(* IEC 61131-3 sources: beebread/doc (part 2) *)

FUNCTION WORD_TO_RANGE : REAL
VAR_INPUT
	X : WORD;
	low : REAL;
	high : REAL;
END_VAR

WORD_TO_RANGE := (high - low) * WORD_TO_REAL(X) * 0.00001525902189669640 + low;
END_FUNCTION

// Commented out for beedance: it uses CHR_TO_STRING, which is commented out.
// FUNCTION LIST_ADD : BOOL
// VAR_INPUT
// 	SEP : BYTE;
// 	INS : STRING(LIST_LENGTH);
// END_VAR
// VAR_IN_OUT
// 	LIST : STRING(LIST_LENGTH);
// END_VAR
// VAR
// 	sx : STRING(1);
// END_VAR
// VAR
// 	INS_work : STRING;
// END_VAR
// (* IEC 61131-3 does not let a POU assign to its inputs, so the body works on copies. *)
// INS_work := INS;
//
// sx := CHR_TO_STRING(SEP);			(* convert separation character to string *)
// INS_work := CONCAT(sx, INS_work);					(* start element with separation character *)
//
// IF LEN(LIST) + LEN(INS_work) > LIST_LENGTH THEN
// 	LIST_ADD := FALSE;					(* return false if element does not fit *)
// ELSE
// 	LIST := CONCAT(LIST, INS_work);
// 	LIST_ADD := TRUE;
// END_IF;
// END_FUNCTION

// Commented out for beedance: it reads or writes the bytes of a STRING through a pointer; a beedance reference (REF_TO) refers to a whole variable of its type.
// FUNCTION LIST_CLEAN : BOOL
// VAR_INPUT
// 	SEP : BYTE;
// END_VAR
// VAR_IN_OUT
// 	LIST : STRING(LIST_LENGTH);
// END_VAR
// VAR
// 	pt : REF_TO ARRAY[1..LIST_LENGTH] OF BYTE;
// 	read : INT := 1;
// 	write : INT := 1;
// 	last: BYTE;
// 	c: BYTE;
// END_VAR
//
// pt := REF(LIST);
//
// FOR read := 1 TO LIST_LENGTH DO
// 	c := pt^[read];								(* read character from list *)
// 	IF c = 0 THEN EXIT;						(* exit the loop if character definbes end of string *)
// 	ELSIF c <> SEP OR sep <> last THEN	(* copy element from read to write position unless a double sep character is present *)
// 		pt^[write] := c;
// 		write := write + 1;
// 	END_IF;
// 	last := c;									(* remember last character *)
// END_FOR;
//
// IF last = SEP THEN write := write - 1; END_IF;		(* if last character is sep then delete empty element at end *)
// IF write <= STRING_LENGTH THEN pt^[write] := 0;	 END_IF;		(* terminate string with 0 *)
//
// LIST_CLEAN := TRUE;						(* retrun TRUE *)
// END_FUNCTION

// Commented out for beedance: it reads or writes the bytes of a STRING through a pointer; a beedance reference (REF_TO) refers to a whole variable of its type.
// FUNCTION LIST_GET : STRING(LIST_LENGTH)
// VAR_INPUT
// 	SEP : BYTE;
// 	POS : INT;
// END_VAR
// VAR_IN_OUT
// 	LIST : STRING(LIST_LENGTH);
// END_VAR
// VAR
// 	i : INT := 1;
// 	o : INT := 1;
// 	pt : REF_TO ARRAY[1..LIST_LENGTH] OF BYTE;
// 	po : REF_TO ARRAY[1..LIST_LENGTH] OF BYTE;
// 	cnt: INT := 0;
// 	c: BYTE;
// END_VAR
//
// pt := REF(LIST);							(* load pointers *)
// po := REF(LIST_GET);
//
// REPEAT
// 	c := pt^[i];
// 	IF cnt = pos THEN						(* copy element to output string *)
// 		IF c = SEP  THEN EXIT; END_IF;		(* next element stop copy and finish *)
// 		po^[o] := c;
// 		o := o + 1;
// 	ELSIF c = SEP THEN
// 		cnt := cnt + 1;
// 	END_IF;
// 	i := i + 1;
// UNTIL
// 	(i = LIST_LENGTH) OR (c = 0)
// END_REPEAT;
// po^[o] := 0;						(* close the output string *)
// END_FUNCTION

// Commented out for beedance: it reads or writes the bytes of a STRING through a pointer; a beedance reference (REF_TO) refers to a whole variable of its type.
// FUNCTION LIST_INSERT : BOOL
// VAR_INPUT
// 	SEP : BYTE;
// 	POS : INT;
// 	INS : STRING(LIST_LENGTH);
// END_VAR
// VAR_IN_OUT
// 	LIST : STRING(LIST_LENGTH);
// END_VAR
// VAR
// 	pt : REF_TO ARRAY[1..LIST_LENGTH] OF BYTE;
// 	read : INT := 1;
// 	cnt : INT := 1;
// 	sx : STRING(1);
// END_VAR
//
// (* load pointers *)
// pt := REF(LIST);
//
// IF LEN(ins) + 1 + LEN(LIST) > LIST_LENGTH THEN
// 	LIST_INSERT := FALSE;
// ELSE
// 	LIST_INSERT := TRUE;
// 	(* search for position *)
// 	WHILE read < LIST_LENGTH DO
// 		IF cnt >= POS THEN
// 			sx := CHR_TO_STRING(SEP);
// 			INS := CONCAT(sx, INS);
// 			LIST := INSERT(LIST, INS, read - 1);
// 			LIST_INSERT := TRUE;
// 			RETURN;
// 		END_IF;
// 		IF pt^[read]  = 0 THEN				(* list is too short add empty element *)
// 			pt^[read] := SEP;
// 			pt^[read + 1] := 0;
// 		END_IF;
// 		read := read + 1;
// 		IF pt^[read] = SEP OR pt^[read] = 0 THEN cnt := cnt + 1; END_IF;
// 	END_WHILE;
// END_IF;
// END_FUNCTION

// Commented out for beedance: it reads or writes the bytes of a STRING through a pointer; a beedance reference (REF_TO) refers to a whole variable of its type.
// FUNCTION LIST_LEN : INT
// VAR_INPUT
// 	SEP : BYTE;
// END_VAR
// VAR_IN_OUT
// 	LIST : STRING(LIST_LENGTH);
// END_VAR
// VAR
// 	pt : REF_TO ARRAY[1..LIST_LENGTH] OF BYTE;
// 	pos: INT := 1;
// 	c: BYTE;
// END_VAR
//
// pt := REF(LIST);
// LIST_LEN := 0;
// REPEAT
// 	c := pt^[pos];
// 	IF c = SEP THEN LIST_LEN := LIST_LEN + 1; END_IF;
// 	pos := pos + 1;
// UNTIL
// 	c = 0 OR pos > LIST_LENGTH
// END_REPEAT;
// END_FUNCTION

// Commented out for beedance: it reads or writes the bytes of a STRING through a pointer; a beedance reference (REF_TO) refers to a whole variable of its type.
// FUNCTION_BLOCK LIST_NEXT
// VAR_INPUT
// 	SEP : BYTE;
// 	RST : BOOL;
// END_VAR
// VAR_IN_OUT
// 	LIST : STRING(LIST_LENGTH);
// END_VAR
// VAR_OUTPUT
// 	LEL : STRING(LIST_LENGTH);
// 	NUL : BOOL;
// END_VAR
// VAR
// 	pos : INT := 1;
// 	pt : REF_TO ARRAY[1..LIST_LENGTH] OF BYTE;
// 	po : REF_TO ARRAY[1..LIST_LENGTH] OF BYTE;
// 	c: BYTE;
// 	write: INT;
// END_VAR
//
// pt := REF(LIST);
// po := REF(LEL);
//
// IF rst THEN
// 	pos := 1;
// END_IF;
//
// IF pt^[pos] = 0 OR pos = LIST_LENGTH THEN
// 	LEL := '';
// 	NUL := TRUE;
// ELSE
// 	NUL := FALSE;
// 	write := 1;
// 	FOR pos := pos + 1 TO LIST_LENGTH DO
// 		c := pt^[pos];
// 		IF c = 0 OR c = SEP THEN
// 			po^[write] := 0;
// 			RETURN;
// 		ELSE
// 			po^[write] := pt^[pos];
// 			write := write + 1;
// 		END_IF;
// 	END_FOR;
// END_IF;
// END_FUNCTION_BLOCK

// Commented out for beedance: it reads or writes the bytes of a STRING through a pointer; a beedance reference (REF_TO) refers to a whole variable of its type.
// FUNCTION LIST_RETRIEVE : STRING(LIST_LENGTH)
// VAR_INPUT
// 	SEP : BYTE;
// 	POS : INT;
// END_VAR
// VAR_IN_OUT
// 	LIST : STRING(LIST_LENGTH);
// END_VAR
// VAR
// 	i :	INT;
// 	o : INT := 1;
// 	w : INT := 1;
// 	pt : REF_TO ARRAY[1..LIST_LENGTH] OF BYTE;
// 	po : REF_TO ARRAY[1..LIST_LENGTH] OF BYTE;
// 	cnt: INT := 0;
// 	c: BYTE;
// END_VAR
//
// (* load pointers *)
// pt := REF(LIST);
// po := REF(LIST_RETRIEVE);
//
// IF pos > 0 THEN
// 	FOR i := 1 TO LIST_LENGTH DO
// 		c := pt^[i];
// 		IF c = 0 THEN
// 			po^[o] := 0;
// 			IF cnt < pos THEN pt^[w + 1] := 0; ELSE pt^[w] := 0; END_IF;
// 			RETURN;
// 		ELSIF cnt = pos AND c <> SEP THEN				(* we have found the element *)
// 			po^[o] := pt^[i];
// 			o := o + 1;
// 		ELSIF cnt >= pos THEN
// 			pt^[w] := c;
// 			w := w + 1;
// 		ELSE
// 			w := i;
// 		END_IF;
// 		IF c = sep THEN cnt := cnt + 1; END_IF;
// 	END_FOR;
// ELSE
// 	LIST_RETRIEVE := '';
// END_IF;
// END_FUNCTION

// Commented out for beedance: it reads or writes the bytes of a STRING through a pointer; a beedance reference (REF_TO) refers to a whole variable of its type.
// FUNCTION LIST_RETRIEVE_LAST : STRING(LIST_LENGTH)
// VAR_INPUT
// 	SEP : BYTE;
// END_VAR
// VAR_IN_OUT
// 	LIST : STRING(LIST_LENGTH);
// END_VAR
// VAR
// 	i :	INT;
// 	last : INT := 1;
// 	pt : REF_TO ARRAY[1..LIST_LENGTH] OF BYTE;
// 	c: BYTE;
// END_VAR
//
// (* load pointers *)
// pt := REF(LIST);
//
// (* search position of last element *)
// FOR i := 1 TO LIST_LENGTH DO
// 	c := pt^[i];
// 	IF c = 0 THEN
// 		EXIT;
// 	ELSIF C = SEP THEN
// 		last := i;
// 	END_IF;
// END_FOR;
// (* return last element of list *)
// LIST_RETRIEVE_LAST := MID(LIST, LIST_LENGTH, last + 1);
// (* terminate list at i *)
// pt^[last] := 0;
// END_FUNCTION

FUNCTION_BLOCK COUNT_BR
VAR_INPUT
	SET : BOOL;
	IN : BYTE;
	UP : BOOL;
	DN : BOOL;
	STEP : BYTE := 1;
	MX : BYTE := 255;
	RST : BOOL;
END_VAR
VAR_OUTPUT
	CNT : BYTE;
END_VAR
VAR
	last_up: BOOL;
	last_dn: BOOL;
END_VAR

IF rst THEN
	cnt := 0;
ELSIF set THEN
	cnt := LIMIT(0,in,mx);
ELSIF up AND NOT last_up THEN
	cnt := INT_TO_BYTE(INC(cnt,step,mx));
ELSIF dn AND NOT last_dn THEN
	cnt := INT_TO_BYTE(inc(cnt,-step,mx));
END_IF;
last_up := up;
last_dn := dn;
END_FUNCTION_BLOCK

FUNCTION_BLOCK COUNT_DR
VAR_INPUT
	SET : BOOL;
	IN : DWORD;
	UP : BOOL;
	DN : BOOL;
	STEP : DWORD := 1;
	MX : DWORD := 16#FFFFFFFF;
	RST : BOOL;
END_VAR
VAR_OUTPUT
	CNT : DWORD;
END_VAR
VAR
	last_up: BOOL;
	last_dn: BOOL;
END_VAR

IF rst THEN
	cnt := 0;
ELSIF set THEN
	cnt := LIMIT(DWORD#0,in,mx);
ELSIF up AND NOT last_up THEN
	IF STEP > ULINT_TO_DWORD((DWORD_TO_ULINT(MX) + 4294967296 - DWORD_TO_ULINT(CNT)) MOD 4294967296) THEN
		CNT := ULINT_TO_DWORD((DWORD_TO_ULINT(CNT) + 4294967296 - DWORD_TO_ULINT(MX) + DWORD_TO_ULINT(STEP) - 1) MOD 4294967296);
	ELSE
		CNT := ULINT_TO_DWORD((DWORD_TO_ULINT(CNT) + DWORD_TO_ULINT(STEP)) MOD 4294967296);
	END_IF;
ELSIF dn AND NOT last_dn THEN
	IF STEP > CNT THEN
		CNT := ULINT_TO_DWORD((DWORD_TO_ULINT(CNT) + 4294967296 - DWORD_TO_ULINT(STEP) + DWORD_TO_ULINT(MX) + 1) MOD 4294967296);
	ELSE
		CNT := ULINT_TO_DWORD((DWORD_TO_ULINT(CNT) + 4294967296 - DWORD_TO_ULINT(STEP)) MOD 4294967296);
	END_IF;
END_IF;
last_up := up;
last_dn := dn;
END_FUNCTION_BLOCK

FUNCTION_BLOCK FF_D2E
VAR_INPUT
	D0 : BOOL;
	D1 : BOOL;
	CLK : BOOL;
	RST : BOOL;
END_VAR
VAR_OUTPUT
	Q0 : BOOL;
	Q1 : BOOL;
END_VAR
VAR
	edge : BOOL;
END_VAR

IF rst THEN
	Q0 := FALSE;
	Q1 := FALSE;
ELSIF clk AND NOT edge THEN
	Q0 := D0;
	Q1 := D1;
END_IF;
edge := CLK;
END_FUNCTION_BLOCK

FUNCTION_BLOCK FF_D4E
VAR_INPUT
	D0 : BOOL;
	D1 : BOOL;
	D2 : BOOL;
	D3 : BOOL;
	CLK : BOOL;
	RST : BOOL;
END_VAR
VAR_OUTPUT
	Q0 : BOOL;
	Q1 : BOOL;
	Q2 : BOOL;
	Q3 : BOOL;
END_VAR
VAR
	edge : BOOL;
END_VAR

IF rst THEN
	Q0 := FALSE;
	Q1 := FALSE;
	Q2 := FALSE;
	Q3 := FALSE;
ELSIF clk AND NOT edge THEN
	Q0 := D0;
	Q1 := D1;
	Q2 := D2;
	Q3 := D3;
END_IF;
edge := CLK;
END_FUNCTION_BLOCK

FUNCTION_BLOCK FF_DRE
VAR_INPUT
	SET : BOOL;
	D : BOOL;
	CLK : BOOL;
	RST : BOOL;
END_VAR
VAR_OUTPUT
	Q : BOOL;
END_VAR
VAR
	edge : BOOL;
END_VAR

IF rst OR set THEN
	Q := NOT rst;
ELSIF clk AND NOT edge THEN
	Q := D;
END_IF;
edge := CLK;
END_FUNCTION_BLOCK

FUNCTION_BLOCK FF_JKE
VAR_INPUT
	SET : BOOL;
	J : BOOL;
	CLK : BOOL;
	K : BOOL;
	RST : BOOL;
END_VAR
VAR_OUTPUT
	Q : BOOL;
END_VAR
VAR
	edge : BOOL;
END_VAR

IF rst OR set THEN
	Q := NOT rst;
ELSIF clk AND NOT edge THEN
	IF J XOR K THEN Q := J;
	ELSE Q := K XOR Q;
	END_IF;
END_IF;
edge := CLK;
END_FUNCTION_BLOCK

FUNCTION_BLOCK FF_RSE
VAR_INPUT
	CS : BOOL;
	CR : BOOL;
	RST : BOOL;
END_VAR
VAR_OUTPUT
	Q : BOOL;
END_VAR
VAR
	es, er : BOOL;
END_VAR

IF rst THEN
	(* asynchronous reset *)
	Q := FALSE;
ELSIF CR AND NOT er THEN
	(* rising edge on CR *)
	Q := FALSE;
ELSIF CS AND NOT es THEN
	(* rising edge on CS *)
	Q := TRUE;
END_IF;

es := CS;
er := CR;
END_FUNCTION_BLOCK

FUNCTION_BLOCK SELECT_8
VAR_INPUT
	E : BOOL;
	SET : BOOL;
	IN : BYTE;
	UP : BOOL;
	DN : BOOL;
	RST : BOOL;
END_VAR
VAR_OUTPUT
	Q0, Q1, Q2, Q3, Q4, Q5, Q6, Q7 : BOOL;
	STATE : INT;
END_VAR
VAR
	last_up: BOOL;
	last_dn : BOOL;
END_VAR

IF rst THEN
	state := 0;
ELSIF set THEN
	state := IN;
ELSIF up AND NOT last_up THEN
	state := inc(state,1,7);
ELSIF dn AND NOT last_dn THEN
	state := inc(state,-1,7);
END_IF;
last_UP := UP;
last_DN := DN;

Q0 := FALSE;
Q1 := FALSE;
Q2 := FALSE;
Q3 := FALSE;
Q4 := FALSE;
Q5 := FALSE;
Q6 := FALSE;
Q7 := FALSE;

IF E THEN
	CASE state OF
		0: Q0 := TRUE;
		1: Q1 := TRUE;
		2: Q2 := TRUE;
		3: Q3 := TRUE;
		4: Q4 := TRUE;
		5: Q5 := TRUE;
		6: Q6 := TRUE;
		7: Q7 := TRUE;
	END_CASE;
END_IF;
END_FUNCTION_BLOCK

FUNCTION_BLOCK SHR_4E
VAR_INPUT
	SET : BOOL;
	D0: BOOL;
	CLK: BOOL;
	RST: BOOL;
END_VAR
VAR_OUTPUT
	Q0: BOOL;
	Q1: BOOL;
	Q2: BOOL;
	Q3: BOOL;
END_VAR
VAR
	trig : R_TRIG;
END_VAR

(* trig.Q signals a rising edge on clk *)
trig(clk := clk);

IF set OR rst THEN
	Q0 := NOT rst;
	Q1 := Q0;
	Q2 := Q0;
	Q3 := Q0;
ELSIF trig.Q THEN
	Q3 := Q2;
	Q2 := Q1;
	Q1 := Q0;
	Q0 := D0;
END_IF;
END_FUNCTION_BLOCK

FUNCTION_BLOCK SHR_4UDE
VAR_INPUT
	SET : BOOL;
	D0: BOOL;
	D3: BOOL;
	CLK: BOOL;
	DN : BOOL;
	RST: BOOL;

END_VAR
VAR_OUTPUT
	Q0: BOOL;
	Q1: BOOL;
	Q2: BOOL;
	Q3: BOOL;
END_VAR
VAR
	trig : R_TRIG;
END_VAR

(* trig.Q signals a rising edge on clk *)
trig(clk := clk);

IF set OR rst THEN
	Q0 := NOT RST;
	Q1 := Q0;
	Q2 := Q0;
	Q3 := Q0;
ELSIF trig.Q THEN
	IF dn THEN
		Q0 := Q1;
		Q1 := Q2;
		Q2 := Q3;
		Q3 := D3;
	ELSE
		Q3 := Q2;
		Q2 := Q1;
		Q1 := Q0;
		Q0 := D0;
	END_IF;
END_IF;
END_FUNCTION_BLOCK

FUNCTION_BLOCK SHR_8PLE
VAR_INPUT
	Din : BOOL;
	Dload : BYTE;
	CLK: BOOL;
	UP: BOOL :=1;
	load : BOOL;
	RST: BOOL;
END_VAR
VAR_OUTPUT
	DOut: BOOL;
END_VAR
VAR
	edge : BOOL :=1;
	register : BYTE;
END_VAR

(* edge detection: clk goes high and edge was high, reset is not active and set is not active *)
IF CLK AND edge AND NOT rst THEN
	edge := FALSE;	(* edge was detected; further edge detection is blocked until edge is true again *)
	(* here is the code for the edge event *)
	IF UP THEN						(*shift up *)
		register := SHL(register,1);
		register.0 := Din;
		Dout := register.7;
	ELSE								(* shift down *);
		register := SHR(register,1);
		register.7 := Din;
		Dout := register.0;
	END_IF;
	IF load THEN							(* the byte on Din will be loaded if load = true *)
		register := Dload;
		IF up THEN Dout := register.7; ELSE Dout := register.0; END_IF;
	END_IF;
END_IF;
IF NOT clk THEN edge := TRUE; END_IF;	(* as soon as clk goes low again, wait for the next edge *)
IF rst THEN									(* if reset is active, reset the output *)
	register := 0;
	Dout := FALSE;
END_IF;
END_FUNCTION_BLOCK

FUNCTION_BLOCK SHR_8UDE
VAR_INPUT
	SET : BOOL;
	D0: BOOL;
	D7: BOOL;
	CLK: BOOL;
	DN : BOOL;
	RST: BOOL;
END_VAR
VAR_OUTPUT
	Q0: BOOL;
	Q1: BOOL;
	Q2: BOOL;
	Q3: BOOL;
	Q4: BOOL;
	Q5: BOOL;
	Q6: BOOL;
	Q7: BOOL;
END_VAR
VAR
	trig : R_TRIG;
END_VAR

(* trig.Q signals a rising edge on clk *)
trig(clk := clk);

IF set OR rst THEN
	Q0 := NOT RST;
	Q1 := Q0;
	Q2 := Q0;
	Q3 := Q0;
	Q4 := Q0;
	Q5 := Q0;
	Q6 := Q0;
	Q7 := Q0;
ELSIF trig.Q THEN
	IF dn THEN
		Q0 := Q1;
		Q1 := Q2;
		Q2 := Q3;
		Q3 := Q4;
		Q4 := Q5;
		Q5 := Q6;
		Q6 := Q7;
		Q7 := D7;
	ELSE
		Q7 := Q6;
		Q6 := Q5;
		Q5 := Q4;
		Q4 := Q3;
		Q3 := Q2;
		Q2 := Q1;
		Q1 := Q0;
		Q0 := D0;
	END_IF;
END_IF;
END_FUNCTION_BLOCK

FUNCTION_BLOCK TOGGLE
VAR_INPUT
	CLK : BOOL;
	rst : BOOL;
END_VAR
VAR_OUTPUT
	Q : BOOL;
END_VAR
VAR
	edge : BOOL;
END_VAR

IF rst THEN
	q := 0;
ELSIF clk AND NOT edge THEN
	Q := NOT Q;
END_IF;
edge := clk;
END_FUNCTION_BLOCK

FUNCTION_BLOCK LTCH
VAR_INPUT
	D : BOOL;
	L : BOOL;
	RST : BOOL;
END_VAR
VAR_OUTPUT
	Q : BOOL;
END_VAR

(* as long as L is true, the latch is transparent and and change of D is transferred to Q *)
(* of course only when there is no asynchronous reset *)
IF rst THEN				(* if asynchronous reset then Q=0 *)
	Q := FALSE;
ELSIF L THEN			(* latch is transparent *)
	Q := D;
END_IF;
END_FUNCTION_BLOCK

FUNCTION_BLOCK LTCH_4
VAR_INPUT
	D0 : BOOL;
	D1 : BOOL;
	D2 : BOOL;
	D3 : BOOL;
	L : BOOL;
	RST : BOOL;
END_VAR
VAR_OUTPUT
	Q0 : BOOL;
	Q1 : BOOL;
	Q2 : BOOL;
	Q3 : BOOL;
END_VAR

(* as long as L is true, the latch is transparent and and change of D is transferred to Q *)
(* of course only when there is no asynchronous reset *)
IF rst THEN			(* if asynchronous reset then Q=0 *)
	Q0 := FALSE;
	Q1 := FALSE;
	Q2 := FALSE;
	Q3 := FALSE;
ELSIF L THEN			(* latch is transparent *)
	Q0 := D0;
	Q1 := D1;
	Q2 := D2;
	Q3 := D3;
END_IF;
END_FUNCTION_BLOCK

FUNCTION_BLOCK STORE_8
VAR_INPUT
	Set : BOOL;
	D0,D1, D2, D3, D4, D5, D6, D7 : BOOL;
	Clr : BOOL;
	Rst : BOOL;
END_VAR
VAR_OUTPUT
	Q0, Q1, Q2, Q3, Q4, Q5, Q6, Q7 : BOOL;
END_VAR
VAR
	edge: BOOL;
END_VAR

IF rst OR set THEN
	q0 := NOT rst;
	q1 := q0;
	q2 := q0;
	q3 := q0;
	q4 := q0;
	q5 := q0;
	q6 := q0;
	q7 := q0;
ELSE
	IF D0 THEN Q0 := TRUE; END_IF;
	IF D1 THEN Q1 := TRUE; END_IF;
	IF D2 THEN Q2 := TRUE; END_IF;
	IF D3 THEN Q3 := TRUE; END_IF;
	IF D4 THEN Q4 := TRUE; END_IF;
	IF D5 THEN Q5 := TRUE; END_IF;
	IF D6 THEN Q6 := TRUE; END_IF;
	IF D7 THEN Q7 := TRUE; END_IF;

	IF clr AND NOT edge THEN
		IF q0 THEN q0 := FALSE;
		ELSIF q1 THEN q1 := FALSE;
		ELSIF q2 THEN q2 := FALSE;
		ELSIF q3 THEN q3 := FALSE;
		ELSIF q4 THEN q4 := FALSE;
		ELSIF q5 THEN q5 := FALSE;
		ELSIF q6 THEN q6 := FALSE;
		ELSE q7 := FALSE;
		END_IF;
	END_IF;
	edge := clr;
END_IF;
END_FUNCTION_BLOCK

FUNCTION BCDC_TO_INT : INT
VAR_INPUT
	IN : BYTE;
END_VAR

BCDC_TO_INT := BYTE_TO_INT(in AND 16#0F) + BYTE_TO_INT(SHR(in,4)) * 10;
END_FUNCTION

FUNCTION BIT_COUNT : INT
VAR_INPUT
	IN : DWORD;
END_VAR
VAR
	IN_work : DWORD;
END_VAR
(* IEC 61131-3 does not let a POU assign to its inputs, so the body works on copies. *)
IN_work := IN;

WHILE IN_work > 0 DO
	IF IN_work.0 THEN Bit_Count := Bit_Count + 1; END_IF;
	IN_work := SHR(IN_work,1);
END_WHILE;
END_FUNCTION

FUNCTION BIT_LOAD_B : BYTE
VAR_INPUT
	IN : BYTE;
	VAL : BOOL;
	POS : INT;
END_VAR
VAR CONSTANT
	dat : BYTE := 1;
END_VAR

IF VAL THEN
	BIT_LOAD_B := in OR SHL(dat,pos);
ELSE
	BIT_LOAD_B := in AND (NOT SHL(dat,pos));
END_IF;
END_FUNCTION

FUNCTION BIT_LOAD_B2 : BYTE
VAR_INPUT
	I : BYTE;
	D : BOOL;
	P : INT;
	N : INT;
END_VAR

IF D THEN
	BIT_LOAD_B2 := ROL(SHR(BYTE#255, 8 - N) OR ROR(i, P), P);
ELSE
	BIT_LOAD_B2 := ROL(SHL(BYTE#255, N) AND ROR(I, P), P);
END_IF;
END_FUNCTION

FUNCTION BIT_LOAD_DW : DWORD
VAR_INPUT
	IN : DWORD;
	VAL : BOOL;
	POS : INT;
END_VAR
VAR CONSTANT
	dat : DWORD := 1;
END_VAR

IF val THEN
	BIT_LOAD_DW := in OR SHL(dat,pos);
ELSE
	BIT_LOAD_DW := in AND (NOT SHL(dat,pos));
END_IF;
END_FUNCTION

FUNCTION BIT_LOAD_DW2 : DWORD
VAR_INPUT
	I : DWORD;
	D : BOOL;
	P : INT;
	N : INT;
END_VAR

IF D THEN
	BIT_LOAD_DW2 := ROL(SHR(DWORD#4294967295, 32 - N) OR ROR(i, P), P);
ELSE
	BIT_LOAD_DW2 := ROL(SHL(DWORD#4294967295, N) AND ROR(I, P), P);
END_IF;
END_FUNCTION

FUNCTION BIT_LOAD_W : WORD
VAR_INPUT
	IN : WORD;
	VAL : BOOL;
	POS : INT;
END_VAR
VAR CONSTANT
	dat : WORD := 1;
END_VAR

IF val THEN
	BIT_LOAD_W := in OR SHL(dat,pos);
ELSE
	BIT_LOAD_W := in AND (NOT SHL(dat,pos));
END_IF;
END_FUNCTION

FUNCTION BIT_LOAD_W2 : WORD
VAR_INPUT
	I : WORD;
	D : BOOL;
	P : INT;
	N : INT;
END_VAR

IF D THEN
	BIT_LOAD_W2 := ROL(SHR(WORD#65535, 16 - N) OR ROR(i, P), P);
ELSE
	BIT_LOAD_W2 := ROL(SHL(WORD#65535, N) AND ROR(I, P), P);
END_IF;
END_FUNCTION

FUNCTION BIT_OF_DWORD : BOOL
VAR_INPUT
	in : DWORD;
	N : INT;
END_VAR

BIT_OF_DWORD := (SHR(in,N) AND 16#00000001) > 0;
END_FUNCTION

FUNCTION BIT_TOGGLE_B : BYTE
VAR_INPUT
	IN : BYTE;
	POS : INT;
END_VAR

BIT_TOGGLE_B := SHL(BYTE#1, POS) XOR IN;
END_FUNCTION

FUNCTION BIT_TOGGLE_DW : DWORD
VAR_INPUT
	IN : DWORD;
	POS : INT;
END_VAR

BIT_TOGGLE_DW := SHL(DWORD#1, POS) XOR IN;
END_FUNCTION

FUNCTION BIT_TOGGLE_W : WORD
VAR_INPUT
	IN : WORD;
	POS : INT;
END_VAR

BIT_TOGGLE_W := SHL(WORD#1, POS) XOR IN;
END_FUNCTION

FUNCTION BYTE_OF_BIT : BYTE
VAR_INPUT
	B0:BOOL;
	B1:BOOL;
	B2:BOOL;
	B3:BOOL;
	B4:BOOL;
	B5:BOOL;
	B6:BOOL;
	B7:BOOL;
END_VAR

Byte_of_bit := SHL(SHL(SHL(SHL(SHL(SHL(SHL(BOOL_TO_BYTE(B7),1) OR BOOL_TO_BYTE(B6),1) OR BOOL_TO_BYTE(B5),1) OR BOOL_TO_BYTE(B4),1)
	OR BOOL_TO_BYTE(B3),1) OR BOOL_TO_BYTE(B2),1) OR BOOL_TO_BYTE(B1),1) OR BOOL_TO_BYTE(B0);
END_FUNCTION

FUNCTION BYTE_OF_DWORD : BYTE
VAR_INPUT
	in : DWORD;
	N : BYTE;
END_VAR

BYTE_OF_DWORD := DWORD_TO_BYTE(SHR(in,SHL(n,3)));
END_FUNCTION

FUNCTION_BLOCK BYTE_TO_BITS
VAR_INPUT
	IN: BYTE;
END_VAR
VAR_OUTPUT
	B0: BOOL;
	B1: BOOL;
	B2: BOOL;
	B3: BOOL;
	B4: BOOL;
	B5: BOOL;
	B6: BOOL;
	B7: BOOL;
END_VAR

B0 := IN.0;
B1 := IN.1;
B2 := IN.2;
B3 := IN.3;
B4 := IN.4;
B5 := IN.5;
B6 := IN.6;
B7 := IN.7;
END_FUNCTION_BLOCK

FUNCTION BYTE_TO_GRAY : BYTE
VAR_INPUT
	IN : BYTE;
END_VAR

BYTE_TO_GRAY := IN XOR SHR(IN,1);
END_FUNCTION

FUNCTION CHECK_PARITY : BOOL
VAR_INPUT
	in : DWORD;
	p : BOOL;
END_VAR
VAR
	in_work : DWORD;
END_VAR
(* IEC 61131-3 does not let a POU assign to its inputs, so the body works on copies. *)
in_work := in;

CHECK_PARITY := NOT p;
WHILE in_work > 0 DO
	CHECK_PARITY := CHECK_PARITY XOR in_work.0 XOR in_work.1 XOR in_work.2 XOR in_work.3;
	in_work := SHR(in_work,4);
END_WHILE;
END_FUNCTION

// Commented out for beedance: it reads the bits of a REAL as a DWORD, or back, through a pointer; a beedance reference (REF_TO) refers to a variable of its own type.
// FUNCTION CHK_REAL : BYTE
// VAR_INPUT
// 	X : REAL;
// END_VAR
// VAR
// 	pt : REF_TO DWORD;
// 	tmp : DWORD;
// END_VAR
//
// pt := REF(X);				(* move real to dword, real_to_dword does not work becasze it treats dword as a number on many systems *)
// tmp := ROL(pt^,1);			(* rotate left foir easy checking, sign will be at lease significant digit *)
// IF tmp < 16#FF000000 THEN
// 	CHK_REAL := 16#00;		(* normalized and denormalized numbers *)
// ELSIF tmp = 16#FF000000 THEN
// 	CHK_REAL := 16#20;		(* X is +infinity see IEEE754 *)
// ELSIF tmp = 16#FF000001 THEN
// 	CHK_REAL := 16#40;		(* X is -infinity see IEEE754 *)
// ELSE
// 	CHK_REAL := 16#80;		(* X is NAN see IEEE754 *)
// END_IF;
// END_FUNCTION

FUNCTION_BLOCK DEC_2
VAR_INPUT
	D: BOOL;
	A: BOOL;
END_VAR
VAR_OUTPUT
	Q0: BOOL;
	Q1: BOOL;
END_VAR

Q0 := D AND NOT A;
Q1 := D AND A;
END_FUNCTION_BLOCK

FUNCTION_BLOCK DEC_4
VAR_INPUT
	D: BOOL;
	A0: BOOL;
	A1: BOOL;
END_VAR
VAR_OUTPUT
	Q0: BOOL;
	Q1: BOOL;
	Q2: BOOL;
	Q3: BOOL;
END_VAR

Q0 := D AND NOT A0 AND NOT A1;
Q1 := D AND A0 AND NOT A1;
Q2 := D AND NOT A0 AND A1;
Q3 := D AND A0 AND A1;
END_FUNCTION_BLOCK

FUNCTION_BLOCK DEC_8
VAR_INPUT
	D: BOOL;
	A0: BOOL;
	A1: BOOL;
	A2: BOOL;
END_VAR
VAR_OUTPUT
	Q0: BOOL;
	Q1: BOOL;
	Q2: BOOL;
	Q3: BOOL;
	Q4: BOOL;
	Q5: BOOL;
	Q6: BOOL;
	Q7: BOOL;
END_VAR
VAR
	X : INT;
END_VAR

X.0 := A0; X.1 := A1; X.2 := A2;

Q0 := FALSE;
Q1 := FALSE;
Q2 := FALSE;
Q3 := FALSE;
Q4 := FALSE;
Q5 := FALSE;
Q6 := FALSE;
Q7 := FALSE;

CASE X OF
	0 : Q0 := D;
	1 : Q1 := D;
	2 : Q2 := D;
	3 : Q3 := D;
	4 : Q4 := D;
	5 : Q5 := D;
	6 : Q6 := D;
	7 : Q7 := D;
END_CASE;
END_FUNCTION_BLOCK

// Commented out for beedance: it reads the bits of a REAL as a DWORD, or back, through a pointer; a beedance reference (REF_TO) refers to a variable of its own type.
// FUNCTION DW_TO_REAL : REAL
// VAR_INPUT
// 	X : DWORD;
// END_VAR
// VAR
// 	pt : REF_TO REAL;
// END_VAR
//
// pt := REF(X);
// DW_TO_REAL := pt^;
// END_FUNCTION

FUNCTION DWORD_OF_BYTE : DWORD
VAR_INPUT
	B3 : BYTE;
	B2 : BYTE;
	B1 : BYTE;
	B0 : BYTE;
END_VAR

DWORD_OF_BYTE := SHL(SHL(SHL(BYTE_TO_DWORD(B3),8) OR BYTE_TO_DWORD(B2),8) OR BYTE_TO_DWORD(B1),8) OR BYTE_TO_DWORD(B0);
END_FUNCTION

FUNCTION DWORD_OF_WORD : DWORD
VAR_INPUT
	W1 : WORD;
	W0 : WORD;
END_VAR

DWORD_OF_WORD := SHL(WORD_TO_DWORD(W1),16) OR WORD_TO_DWORD(W0);
END_FUNCTION

FUNCTION GRAY_TO_BYTE : BYTE
VAR_INPUT
	IN : BYTE;
END_VAR

GRAY_TO_BYTE := SHR(IN,4) XOR IN;
GRAY_TO_BYTE := SHR(GRAY_TO_BYTE,2) XOR GRAY_TO_BYTE;
GRAY_TO_BYTE := SHR(GRAY_TO_BYTE,1) XOR GRAY_TO_BYTE;
END_FUNCTION

FUNCTION INT_TO_BCDC : BYTE
VAR_INPUT
	IN : INT;
END_VAR

INT_TO_BCDC := SHL(INT_TO_BYTE(IN / INT#10),4) OR INT_TO_BYTE(in MOD INT#10);
END_FUNCTION

FUNCTION MUX_2 : BOOL
VAR_INPUT
	D0: BOOL;
	D1: BOOL;
	A0: BOOL;
END_VAR

MUX_2 := SEL(A0, D0, D1);
END_FUNCTION

FUNCTION MUX_4 : BOOL
VAR_INPUT
	D0: BOOL;
	D1: BOOL;
	D2: BOOL;
	D3: BOOL;
	A0: BOOL;
	A1: BOOL;
END_VAR

IF A1 THEN
	MUX_4 := SEL(A0, D2, D3);
ELSE
	MUX_4 := SEL(A0, D0, D1);
END_IF;
END_FUNCTION

FUNCTION PARITY : BOOL
VAR_INPUT
	in : DWORD;
END_VAR
VAR
	in_work : DWORD;
END_VAR
(* IEC 61131-3 does not let a POU assign to its inputs, so the body works on copies. *)
in_work := in;

WHILE in_work > 0 DO
	PARITY := PARITY XOR in_work.0 XOR in_work.1 XOR in_work.2 XOR in_work.3;
	in_work := SHR(in_work,4);
END_WHILE;
END_FUNCTION

// Commented out for beedance: it reads the bits of a REAL as a DWORD, or back, through a pointer; a beedance reference (REF_TO) refers to a variable of its own type.
// FUNCTION REAL_TO_DW : DWORD
// VAR_INPUT
// 	X : REAL;
// END_VAR
// VAR
// 	pt : REF_TO DWORD;
// END_VAR
//
// pt := REF(X);
// REAL_TO_DW := pt^;
// END_FUNCTION

FUNCTION REFLECT : DWORD
VAR_INPUT
	D : DWORD;
	L : INT;
END_VAR
VAR
	i : INT;
END_VAR
VAR
	D_work : DWORD;
END_VAR
(* IEC 61131-3 does not let a POU assign to its inputs, so the body works on copies. *)
D_work := D;

REFLECT := 0;
FOR i := 1 TO L DO
	REFLECT := SHL(REFLECT, 1) OR BOOL_TO_DWORD(D_work.0);
	D_work := SHR(D_work, 1);
END_FOR;
REFLECT := REFLECT OR SHL(D_work, L);
END_FUNCTION

FUNCTION REVERSE : BYTE
VAR_INPUT
	IN : BYTE;
END_VAR

(* new code donated by rebler wolfgang *)
REVERSE := ROR(in,1) AND 2#10001000 OR ROL(in,1) AND 2#00010001 OR ROR(in,3) AND 2#01000100 OR ROL(in,3) AND 2#00100010;
END_FUNCTION

FUNCTION SHL1 : DWORD
VAR_INPUT
	IN : DWORD;
	N : INT;
END_VAR
VAR CONSTANT
	temp : DWORD := 16#FFFF_FFFF;
END_VAR

SHL1 := SHR(temp,32-N) OR SHL(IN,N);
END_FUNCTION

FUNCTION SHR1 : DWORD
VAR_INPUT
	IN : DWORD;
	N : INT;
END_VAR
VAR CONSTANT
	temp : DWORD := 16#FFFF_FFFF;
END_VAR

SHR1 := SHL(temp,32-N) OR SHR(IN,N);
END_FUNCTION

FUNCTION SWAP_BYTE : WORD
VAR_INPUT
	IN : WORD;
END_VAR

SWAP_BYTE := ROL(in,8);
END_FUNCTION

FUNCTION SWAP_BYTE2 : DWORD
VAR_INPUT
	IN : DWORD;
END_VAR

Swap_Byte2 := (ROR(in,8) AND 16#FF00FF00) OR (ROL(in,8) AND 16#00FF00FF);
END_FUNCTION

FUNCTION WORD_OF_BYTE : WORD
VAR_INPUT
	B1 : BYTE;
	B0 : BYTE;
END_VAR

WORD_OF_BYTE := SHL(BYTE_TO_WORD(B1),8) OR BYTE_TO_WORD(B0);
END_FUNCTION

FUNCTION WORD_OF_DWORD : WORD
VAR_INPUT
	in : DWORD;
	N : BYTE;
END_VAR

WORD_OF_DWORD := DWORD_TO_WORD(SHR(in,SHL(n,4)));
END_FUNCTION

FUNCTION_BLOCK A_TRIG
VAR_INPUT
	IN : REAL;
	RES : REAL;
END_VAR
VAR_OUTPUT
	Q : BOOL;
	D : REAL;
END_VAR
VAR
	last_in : REAL;
END_VAR

D := IN - LAST_IN;
Q := ABS(D) > res;
IF Q THEN last_in := IN; END_IF;
D := IN - LAST_IN;
END_FUNCTION_BLOCK

FUNCTION_BLOCK B_TRIG
VAR_INPUT
	CLK : BOOL;
END_VAR
VAR_OUTPUT
	Q : BOOL;
END_VAR
VAR
	edge : BOOL;
END_VAR

Q := clk XOR edge;
edge := CLK;
END_FUNCTION_BLOCK

FUNCTION_BLOCK CLICK_CNT
VAR_INPUT
	IN : BOOL;
	N : INT;
	TC : TIME;
END_VAR
VAR_OUTPUT
	Q : BOOL;
END_VAR
VAR
	tx : TP;
	edge: BOOL;
	cnt: INT := -1;
END_VAR

(* Q shall only be active for one cycle only *)
Q := FALSE;

IF in AND NOT edge AND NOT tx.q THEN
	(* a rising edge on in sets the counter to 0 *)
	cnt := 0;
ELSIF tx.Q AND NOT IN AND edge THEN
	(* count falling edges when tp.q is true *)
	cnt := cnt + 1;
ELSIF NOT tx.Q THEN
	Q := cnt = N;
	cnt := -1;
END_IF;

(* remember the status of IN *)
edge := IN;
tx(in := IN, pt := TC);
END_FUNCTION_BLOCK

FUNCTION_BLOCK CLICK_DEC
VAR_INPUT
	IN : BOOL;
	TC : TIME;
END_VAR
VAR_OUTPUT
	Q0, Q1, Q2, Q3 : BOOL;
END_VAR
VAR
	tx : TP;
	edge: BOOL;
	cnt: INT := -1;
END_VAR

(* Q shall only be active for one cycle only *)
IF in = FALSE THEN
	Q0 := FALSE;
	Q1 := FALSE;
	Q2:= FALSE;
	Q3 := FALSE;
END_IF;

IF in AND NOT edge AND NOT tx.q THEN
	(* a rising edge on in sets the counter to 0 *)
	cnt := 0;
ELSIF tx.Q AND NOT IN AND edge THEN
	(* count falling edges when tp.q is true *)
	cnt := cnt + 1;
ELSIF NOT tx.Q THEN
	CASE cnt OF
		0 : Q0 := TRUE;
		1 : Q1 := TRUE;
		2 : Q2 := TRUE;
		3 : Q3 := TRUE;
	END_CASE;
	cnt := -1;
END_IF;

(* remember the status of IN *)
edge := IN;
tx(in := IN, pt := TC);
END_FUNCTION_BLOCK

FUNCTION_BLOCK CLK_DIV
VAR_INPUT
	clk : BOOL;
	rst: BOOL;
END_VAR
VAR_OUTPUT
	Q0 : BOOL;
	Q1 : BOOL;
	Q2 : BOOL;
	Q3 : BOOL;
	Q4 : BOOL;
	Q5 : BOOL;
	Q6 : BOOL;
	Q7 : BOOL;
END_VAR
VAR
	cnt: BYTE;
END_VAR

IF rst THEN
	cnt:= 0;
	Q0 := 0;
	Q1 := 0;
	Q2 := 0;
	Q3 := 0;
	Q4 := 0;
	Q5 := 0;
	Q6 := 0;
	Q7 := 0;
ELSIF clk THEN
	cnt := ULINT_TO_BYTE((BYTE_TO_ULINT(cnt) + 1) MOD 256);
	Q0 := cnt.0;
	Q1 := cnt.1;
	Q2 := cnt.2;
	Q3 := cnt.3;
	Q4 := cnt.4;
	Q5 := cnt.5;
	Q6 := cnt.6;
	Q7 := cnt.7;
END_IF;
END_FUNCTION_BLOCK

FUNCTION_BLOCK CLK_N
VAR_INPUT
	N : INT;
END_VAR
VAR_OUTPUT
	Q : BOOL;
END_VAR
VAR
	edge : BOOL;
	stime: DWORD;
	clk: BOOL;
END_VAR

stime := SHR(T_PLC_MS(),N);
clk := stime.0;
Q := clk XOR edge;
edge := CLK;
END_FUNCTION_BLOCK

FUNCTION_BLOCK CLK_PRG
VAR_INPUT
	PT : TIME := t#10ms;
END_VAR
VAR_OUTPUT
	Q : BOOL;
END_VAR
VAR
	init : BOOL;
	last : TIME;
	tx: TIME;
END_VAR

(* read system time *)
tx := DWORD_TO_TIME(T_PLC_MS());

(* initialize on startup *)
IF NOT init THEN
	init := TRUE;
	last := tx - pt;
END_IF;

(* generate output pulse when next_pulse is reached *)
Q := tx - last >= pt;
IF Q THEN last := tx; END_IF;
END_FUNCTION_BLOCK

FUNCTION_BLOCK CLK_PULSE
VAR_INPUT
	PT : TIME;
	N : INT;
	RST : BOOL ;
END_VAR
VAR_OUTPUT
	Q : BOOL;
	CNT : INT;
	RUN : BOOL;
END_VAR
VAR
	tx, tn: DWORD;
	init: BOOL;
END_VAR

tx := T_PLC_MS();		(* read system *)
Q := FALSE;				(* reset Q we generate pulses only for one cycle *)
RUN := CNT < N;

IF NOT init OR RST THEN
	init := TRUE;
	CNT := 0;
	tn := ULINT_TO_DWORD((DWORD_TO_ULINT(tx) + 4294967296 - DWORD_TO_ULINT(TIME_TO_DWORD(PT))) MOD 4294967296);
	RUN := FALSE;
ELSIF (cnt < N OR N = 0) AND ULINT_TO_DWORD((DWORD_TO_ULINT(tx) + 4294967296 - DWORD_TO_ULINT(tn)) MOD 4294967296) >= TIME_TO_DWORD(PT) THEN		(* generate a pulse *)
	CNT := CNT + 1;
	Q := TRUE;
	tn := ULINT_TO_DWORD((DWORD_TO_ULINT(tn) + TIME_TO_ULINT(PT)) MOD 4294967296);
END_IF;
END_FUNCTION_BLOCK

FUNCTION_BLOCK CYCLE_4
VAR_INPUT
	E : BOOL := TRUE;
	T0, T1, T2, T3 : TIME;
	S0 : BOOL;
	SX : INT;
	SL : BOOL;
END_VAR
VAR_OUTPUT
	STATE : INT;
END_VAR
VAR
	tx : TIME;
	last : TIME;
	init: BOOL;
END_VAR
VAR
	SL_work : BOOL;
END_VAR
(* IEC 61131-3 does not let a POU assign to its inputs, so the body works on copies. *)
SL_work := SL;

(* read system timer *)
tx := DWORD_TO_TIME(T_PLC_MS());
(* init on first cycle *)
IF NOT init THEN
	init := TRUE;
	last := tx;
END_IF;

IF E THEN
	IF SL_work THEN
		(* when sx > 0 then the state sx is forced to start *)
		state:= LIMIT(0,SX,3);
		last := tx;
		(* this is to avoid to reset sx from the calling programm it does work fine on codesys but i am not sure about other systems, because we are writing to an input *)
		SL_work := FALSE;
	ELSE
		CASE state OF
			0 :	(* wait for T0 and switch to next cycle *)
				IF tx - last >= T0 THEN
					state := 1;
					last := tx;
				END_IF;
			1 : (* wait for T1 over 1st cycle *)
				IF tx - last >= T1 THEN
					state := 2;
					last := tx;
				END_IF;
			2 : (* wait for T1 over 1st cycle *)
				IF tx - last >= T2 THEN
					state := 3;
					last := tx;
				END_IF;
			3 : (* wait for T2 over 2nd cycle *)
				IF tx - last >= T3 THEN
					IF S0 THEN State := 0; END_IF; (* if S0 is false, the sequence stops at state 3 *)
					last := tx;
				END_IF;
		END_CASE;
	END_IF;
ELSE
	state := 0;
	last := tx;
END_IF;
END_FUNCTION_BLOCK

FUNCTION_BLOCK D_TRIG
VAR_INPUT
	in : DWORD;
END_VAR
VAR_OUTPUT
	Q : BOOL;
	X : DWORD;
END_VAR
VAR
	last_in : DWORD;
END_VAR

Q := in <> last_in;
X := ULINT_TO_DWORD((DWORD_TO_ULINT(in) + 4294967296 - DWORD_TO_ULINT(last_in)) MOD 4294967296);
last_in := in;
END_FUNCTION_BLOCK

FUNCTION_BLOCK GEN_BIT
VAR_INPUT
	in0 : DWORD;
	in1 : DWORD;
	in2 : DWORD;
	in3 : DWORD;
	clk : BOOL;
	steps : INT;
	rep : INT;
	rst : BOOL;
END_VAR
VAR_OUTPUT
	Q0 :BOOL;
	Q1 :BOOL;
	Q2 :BOOL;
	Q3 :BOOL;
	cnt : INT;
	run : BOOL;
END_VAR
VAR
	r0: DWORD;
	r1: DWORD;
	r2: DWORD;
	r3: DWORD;
	rx : INT := 1;
END_VAR

(* check if number of runs is finished or rep = 0 which means continuous *)

IF clk AND NOT rst THEN
	run := (rep = 0) OR (rx <= rep);
	IF run THEN
		(* check for step counter reached and reset to 0 if cnt = steps *)
		IF cnt = steps THEN
			cnt := 0;
		END_IF;

		(* when cnt = 0 then reload the inputs into the registers *)
		IF cnt = 0 THEN
			r0 := in0;
			r1 := in1;
			r2 := in2;
			r3 := in3;
		END_IF;

		(* when cnt < steps, shift the lowest bits to the outputs *)
		IF (cnt < steps) THEN
			Q0 := r0.0;
			Q1 := r1.0;
			Q2 := r2.0;
			Q3 := r3.0;
			r0 := SHR(r0,1);
			r1 := SHR(r1,1);
			r2 := SHR(r2,1);
			r3 := SHR(r3,1);
		END_IF;

		(* increment the step counter *)
		cnt := cnt +1;
		IF (cnt = steps) AND (rep <> 0) THEN rx := rx +1; END_IF;
		IF (rx > rep) AND (rep <> 0) THEN run := FALSE; END_IF;
	END_IF;
ELSE
	IF rst THEN
		run := FALSE;
		Q0 := FALSE;
		Q1 := FALSE;
		Q2 := FALSE;
		Q3 := FALSE;
		r0 := 0;
		r1 := 0;
		r2 := 0;
		r3 := 0;
		cnt := 0;
		rx := 1;
	END_IF;
END_IF;
END_FUNCTION_BLOCK

FUNCTION_BLOCK GEN_SQ
VAR_INPUT
	PT : TIME;
END_VAR
VAR_OUTPUT
	Q : BOOL;
END_VAR
VAR
	tn: DWORD;
	tx: DWORD;
	init : BOOL;
END_VAR

(* read system time *)
tx := T_PLC_MS();

IF NOT init THEN
	init := TRUE;
	tn := tx;
	Q := TRUE;
ELSIF ULINT_TO_DWORD((DWORD_TO_ULINT(tx) + 4294967296 - DWORD_TO_ULINT(tn)) MOD 4294967296) >= SHR(TIME_TO_DWORD(PT),1) THEN
	Q := NOT Q;
	tn := ULINT_TO_DWORD((DWORD_TO_ULINT(tn) + DWORD_TO_ULINT(SHR(TIME_TO_DWORD(pt),1))) MOD 4294967296);
END_IF;
END_FUNCTION_BLOCK

FUNCTION_BLOCK SCHEDULER
VAR_INPUT
	E0 : BOOL;
	E1 : BOOL;
	E2 : BOOL;
	E3 : BOOL;
END_VAR
VAR_INPUT CONSTANT
	T0, T1, T2, T3 : TIME;
END_VAR
VAR_OUTPUT
	Q0, Q1, Q2, Q3 : BOOL;
END_VAR
VAR
	init : BOOL;
	s0, s1, s2, s3 : TIME;
	tx : TIME;
	c : INT;
END_VAR

(* read system_time *)
tx := DWORD_TO_TIME(T_PLC_MS());

IF NOT init THEN
	init := TRUE;
	s0 := tx - T0;
	s1 := tx - T1;
	s2 := tx - T2;
	s3 := tx - T3;
END_IF;

Q0 := FALSE;
Q1 := FALSE;
Q2 := FALSE;
Q3 :=FALSE;

CASE c OF
	0: 	IF tx - s0 >= T0 THEN
			Q0 := E0;
			s0 := tx;
		END_IF;
		c := 1;
	1: 	IF tx - s1 >= T1 THEN
			Q1 := E1;
			s1 := tx;
		END_IF;
		c := 2;
	2: 	IF tx - s2 >= T2 THEN
			Q2 := E2;
			s2 := tx;
		END_IF;
		c := 3;
	3: 	IF tx - s3 >= T3 THEN
			Q3 := E3;
			s3 := tx;
		END_IF;
		c := 0;
END_CASE;
END_FUNCTION_BLOCK

FUNCTION_BLOCK SCHEDULER_2
VAR_INPUT
	E0 : BOOL;
	E1 : BOOL;
	E2 : BOOL;
	E3 : BOOL;
END_VAR
VAR_INPUT CONSTANT
	C0, C1, C2, C3 : UINT;
	O0, O1, O2, O3 : UINT;
END_VAR
VAR_OUTPUT
	Q0, Q1, Q2, Q3 : BOOL;
END_VAR
VAR
	sx : UINT;
END_VAR

Q0 := E0 AND (sx MOD C0 - O0 = 0);
Q1 := E1 AND (sx MOD C1 - O1 = 0);
Q2 := E2 AND (sx MOD C2 - O2 = 0);
Q3 := E3 AND (sx MOD C3 - O3 = 0);

(* increment cycle counter every cycle *)
sx := sx + 1;
END_FUNCTION_BLOCK

FUNCTION_BLOCK SEQUENCE_4
VAR_INPUT
	in0 : BOOL := TRUE;
	in1 : BOOL := TRUE;
	in2 : BOOL := TRUE;
	in3 : BOOL := TRUE;
	start : BOOL;
	rst : BOOL;
	wait0 : TIME;
	delay0 : TIME;
	wait1 : TIME;
	delay1 : TIME;
	wait2 : TIME;
	delay2 : TIME;
	wait3 : TIME;
	delay3 : TIME;
END_VAR
VAR_INPUT CONSTANT
	stop_on_error : BOOL;
END_VAR
VAR_OUTPUT
	Q0 : BOOL;
	Q1 : BOOL;
	Q2 : BOOL;
	Q3 : BOOL;
	QX : BOOL;
	run: BOOL;
	step : INT := -1;
	status : BYTE;
END_VAR
VAR
	last : TIME;
	edge : BOOL;
	tx: TIME;
	init: BOOL;
END_VAR

(* read sps timer *)
tx := DWORD_TO_TIME(T_PLC_MS());

(* initialize on startup *)
IF NOT init THEN
	last := tx;
	init := TRUE;
	status := 110;
END_IF;

(* asynchronous reset *)
IF rst THEN
	step := -1;
	Q0 := 0;
	Q1 := 0;
	Q2 := 0;
	Q3 := 0;
	status := 110;
	run := 0;

(* edge on start input restarts the sequencer *)
ELSIF start AND NOT edge THEN
	step := 0;
	last := tx;
	status := 111;
	Q0 := 0;
	Q1 := 0;
	Q2 := 0;
	Q3 := 0;
	run := 1;
END_IF;
edge := start;

(* check if stop on status is necessary *)
IF status > 0 AND status < 100 AND stop_on_error THEN RETURN; END_IF;

(* sequence is running *)
IF run AND step = 0 THEN
	IF NOT q0 AND in0 AND tx - last <= wait0 THEN
		Q0 := TRUE;
		last := tx;
	ELSIF NOT q0 AND tx - last > wait0 THEN
		status := 1;
		run := FALSE;
	ELSIF q0 AND tx - last >= delay0 THEN
		step := 1;
		last := tx;
	END_IF;
END_IF;
IF run AND step = 1 THEN
	IF NOT q1 AND in1 AND tx - last <= wait1 THEN
		Q0 := FALSE;
		Q1 := TRUE;
		last := tx;
	ELSIF NOT q1 AND Tx - last > wait1 THEN
		status := 2;
		q0 := FALSE;
		run := FALSE;
	ELSIF q1 AND tx - last >= delay1 THEN
		step := 2;
		last := tx;
	END_IF;
END_IF;
IF run AND step = 2 THEN
	IF NOT q2 AND in2 AND tx - last <= wait2 THEN
		Q1 := FALSE;
		Q2 := TRUE;
		last := tx;
	ELSIF NOT q2 AND Tx - last > wait2 THEN
		status := 3;
		q1 := FALSE;
		run := FALSE;
	ELSIF q2 AND tx - last >= delay2 THEN
		step := 3;
		last := tx;
	END_IF;
END_IF;
IF run AND step = 3 THEN
	IF NOT q3 AND in3 AND tx - last <= wait3 THEN
		Q2 := FALSE;
		Q3 := TRUE;
		last := tx;
	ELSIF NOT q3 AND Tx - last > wait3 THEN
		status := 4;
		q2 := FALSE;
		run := FALSE;
	ELSIF q3 AND tx - last >= delay3 THEN
		step := -1;
		q3 := FALSE;
		run := FALSE;
		status := 110;
	END_IF;
END_IF;
QX := q0 OR q1 OR q2 OR q3;
END_FUNCTION_BLOCK

FUNCTION_BLOCK SEQUENCE_64
VAR_INPUT
	START : BOOL;
	SMAX : INT;
	PROG : ARRAY[0..63]OF TIME;
	RST : BOOL;
END_VAR
VAR_OUTPUT
	STATE : INT := -1;
	TRIG : BOOL;
END_VAR
VAR
	tx : TIME;
	edge: BOOL;
	last: TIME;
END_VAR

(* read system timer *)
tx := DWORD_TO_TIME(T_PLC_MS());
TRIG := FALSE;

IF RST THEN
	STATE := -1;

(* start sequence *)
ELSIF START AND NOT edge THEN
	STATE := 0;
	last := tx;
	TRIG := TRUE;

(* sequence generator *)
ELSIF (STATE >= 0) THEN
	IF (tx - last) >= PROG[STATE] THEN
		STATE := INC2(STATE, 1, -1, SMAX);
		last := tx;
		TRIG := TRUE;
	END_IF;
END_IF;

edge := START;
END_FUNCTION_BLOCK

FUNCTION_BLOCK SEQUENCE_8
VAR_INPUT
	in0 : BOOL := TRUE;
	in1 : BOOL := TRUE;
	in2 : BOOL := TRUE;
	in3 : BOOL := TRUE;
	in4 : BOOL := TRUE;
	in5 : BOOL := TRUE;
	in6 : BOOL := TRUE;
	in7 : BOOL := TRUE;
	start : BOOL;
	rst : BOOL;
	wait0 : TIME;
	delay0 : TIME;
	wait1 : TIME;
	delay1 : TIME;
	wait2 : TIME;
	delay2 : TIME;
	wait3 : TIME;
	delay3 : TIME;
	wait4 : TIME;
	delay4 : TIME;
	wait5 : TIME;
	delay5 : TIME;
	wait6 : TIME;
	delay6 : TIME;
	wait7 : TIME;
	delay7 : TIME;
END_VAR
VAR_INPUT CONSTANT
	stop_on_error : BOOL;
END_VAR
VAR_OUTPUT
	Q0 : BOOL;
	Q1 : BOOL;
	Q2 : BOOL;
	Q3 : BOOL;
	Q4 : BOOL;
	Q5 : BOOL;
	Q6 : BOOL;
	Q7 : BOOL;
	QX : BOOL;
	run: BOOL;
	step : INT := -1;
	status : BYTE;
END_VAR
VAR
	last : TIME;
	edge : BOOL;
	tx: TIME;
	init: BOOL;
END_VAR

(* read sps timer *)
tx := DWORD_TO_TIME(T_PLC_MS());

(* initialize on startup *)
IF NOT init THEN
	last := tx;
	init := TRUE;
	status := 110;
END_IF;

(* asynchronous reset *)
IF rst THEN
	step := -1;
	Q0 := 0;
	Q1 := 0;
	Q2 := 0;
	Q3 := 0;
	Q4 := 0;
	Q5 := 0;
	Q6 := 0;
	Q7 := 0;
	status := 110;
	run := 0;

(* edge on start input restarts the sequencer *)
ELSIF start AND NOT edge THEN
	step := 0;
	last := tx;
	status := 111;
	Q0 := 0;
	Q1 := 0;
	Q2 := 0;
	Q3 := 0;
	Q4 := 0;
	Q5 := 0;
	Q6 := 0;
	Q7 := 0;
	run := 1;
END_IF;
edge := start;

(* check if stop on error is necessary *)
IF status > 0 AND status < 100 AND stop_on_error THEN RETURN; END_IF;

(* sequence is running *)
IF run AND step = 0 THEN
	IF NOT q0 AND in0 AND tx - last <= wait0 THEN
		Q0 := TRUE;
		last := tx;
	ELSIF NOT q0 AND tx - last > wait0 THEN
		status := 1;
		run := FALSE;
	ELSIF q0 AND tx - last >= delay0 THEN
		step := 1;
		last := tx;
	END_IF;
END_IF;
IF run AND step = 1 THEN
	IF NOT q1 AND in1 AND tx - last <= wait1 THEN
		Q0 := FALSE;
		Q1 := TRUE;
		last := tx;
	ELSIF NOT q1 AND Tx - last > wait1 THEN
		status := 2;
		q0 := FALSE;
		run := FALSE;
	ELSIF q1 AND tx - last >= delay1 THEN
		step := 2;
		last := tx;
	END_IF;
END_IF;
IF run AND step = 2 THEN
	IF NOT q2 AND in2 AND tx - last <= wait2 THEN
		Q1 := FALSE;
		Q2 := TRUE;
		last := tx;
	ELSIF NOT q2 AND Tx - last > wait2 THEN
		status := 3;
		q1 := FALSE;
		run := FALSE;
	ELSIF q2 AND tx - last >= delay2 THEN
		step := 3;
		last := tx;
	END_IF;
END_IF;
IF run AND step = 3 THEN
	IF NOT q3 AND in3 AND tx - last <= wait3 THEN
		Q2 := FALSE;
		Q3 := TRUE;
		last := tx;
	ELSIF NOT q3 AND Tx - last > wait3 THEN
		status := 4;
		q2 := FALSE;
		run := FALSE;
	ELSIF q3 AND tx - last >= delay3 THEN
		step := 4;
		last := tx;
	END_IF;
END_IF;
IF run AND step = 4 THEN
	IF NOT q4 AND in4 AND tx - last <= wait4 THEN
		Q3 := FALSE;
		Q4 := TRUE;
		last := tx;
	ELSIF NOT q4 AND Tx - last > wait4 THEN
		status := 5;
		q3 := FALSE;
		run := FALSE;
	ELSIF q4 AND tx - last >= delay4 THEN
		step := 5;
		last := tx;
	END_IF;
END_IF;
IF run AND step = 5 THEN
	IF NOT q5 AND in5 AND tx - last <= wait5 THEN
		Q4 := FALSE;
		Q5 := TRUE;
		last := tx;
	ELSIF NOT q5 AND Tx - last > wait5 THEN
		status := 6;
		q4 := FALSE;
		run := FALSE;
	ELSIF q5 AND tx - last >= delay5 THEN
		step := 6;
		last := tx;
	END_IF;
END_IF;
IF run AND step = 6 THEN
	IF NOT q6 AND in6 AND tx - last <= wait6 THEN
		Q5 := FALSE;
		Q6 := TRUE;
		last := tx;
	ELSIF NOT q6 AND Tx - last > wait6 THEN
		status := 7;
		q5 := FALSE;
		run := FALSE;
	ELSIF q6 AND tx - last >= delay6 THEN
		step := 7;
		last := tx;
	END_IF;
END_IF;
IF run AND step = 7 THEN
	IF NOT q7 AND in7 AND tx - last <= wait7 THEN
		Q6 := FALSE;
		Q7 := TRUE;
		last := tx;
	ELSIF NOT q7 AND Tx - last > wait7 THEN
		status := 8;
		q6 := FALSE;
		run := FALSE;
	ELSIF q7 AND tx - last >= delay7 THEN
		step := -1;
		Q7 := FALSE;
		Run := FALSE;
		status := 110;
	END_IF;
END_IF;
QX := q0 OR q1 OR q2 OR q3 OR q4 OR q5 OR q6 OR q7;
END_FUNCTION_BLOCK

FUNCTION_BLOCK TMAX
VAR_INPUT
	IN : BOOL;
	PT : TIME;
END_VAR
VAR_OUTPUT
	Q : BOOL;
	Z : BOOL;
END_VAR
VAR
	tx : TIME;
	start : TIME;
	last_in: BOOL;
END_VAR

(* read system timer *)
tx := DWORD_TO_TIME(T_PLC_MS());

Z := FALSE;

IF NOT in THEN
	Q := FALSE;
ELSIF IN AND NOT last_in THEN
	Q := TRUE;
	start := tx;
ELSIF (tx - start >= PT) AND Q THEN
	Q := FALSE;
	Z := TRUE;
END_IF;

last_in := IN;
END_FUNCTION_BLOCK

FUNCTION_BLOCK TMIN
VAR_INPUT
	IN : BOOL;
	PT : TIME;
END_VAR
VAR_OUTPUT
	Q : BOOL;
END_VAR
VAR
	pm : TP;
END_VAR

pm(in := IN, PT := PT);
Q := IN OR pm.Q;
END_FUNCTION_BLOCK

FUNCTION_BLOCK TOF_1
VAR_INPUT
	IN : BOOL;
	PT : TIME;
	RST : BOOL;
END_VAR
VAR_OUTPUT
	Q : BOOL;
END_VAR
VAR
	tx : TIME;
	start : TIME;
END_VAR

(* read system timer *)
tx := DWORD_TO_TIME(T_PLC_MS());

IF RST THEN
	Q := FALSE;
ELSIF IN THEN
	Q := TRUE;
	start := tx;
ELSIF tx - start >= PT THEN
	Q := FALSE;
END_IF;
END_FUNCTION_BLOCK

FUNCTION_BLOCK TONOF
VAR_INPUT
	IN : BOOL;
	  T_ON,T_OFF : TIME;
END_VAR
VAR_OUTPUT
	Q : BOOL;
END_VAR
VAR
   X : TON;
   old: BOOL;
   mode: BOOL;
END_VAR

IF IN XOR old THEN
  X(IN := FALSE, PT := SEL(IN,T_OFF,T_ON));
  mode := IN;
  old := IN;
END_IF;
X(IN := TRUE);
IF X.Q THEN Q := mode;END_IF;
END_FUNCTION_BLOCK

FUNCTION_BLOCK TP_1
VAR_INPUT
	IN : BOOL;
	PT : TIME;
	RST : BOOL;
END_VAR
VAR_OUTPUT
	Q : BOOL;
END_VAR
VAR
	tx : TIME;
	start : TIME;
	ix : BOOL;
END_VAR

(* read system timer *)
tx := DWORD_TO_TIME(T_PLC_MS());

IF RST THEN
	Q := FALSE;
ELSIF IN AND NOT ix THEN
	Q := TRUE;
	start := tx;
ELSIF tx - start >= PT THEN
	Q := FALSE;
END_IF;

ix:= IN;
END_FUNCTION_BLOCK

FUNCTION_BLOCK TP_1D
VAR_INPUT
	IN : BOOL;
	PT1 : TIME;
	PTD : TIME;
	RST : BOOL;
END_VAR
VAR_OUTPUT
	Q : BOOL;
	W : BOOL;
END_VAR
VAR
	tx : TIME;
	start: TIME;
	ix: BOOL;
END_VAR
VAR
	IN_work : BOOL;
	RST_work : BOOL;
END_VAR
(* IEC 61131-3 does not let a POU assign to its inputs, so the body works on copies. *)
IN_work := IN;
RST_work := RST;

(* read system timer *)
tx := DWORD_TO_TIME(T_PLC_MS());

IF RST_work THEN
	Q := FALSE;
	RST_work := FALSE;
	W := FALSE;
ELSIF W THEN
	IF tx - start >= PTD THEN
		W := FALSE;
	END_IF;
ELSIF IN_work AND NOT ix THEN
	Q := TRUE;
	start := tx;
	IN_work := FALSE;
ELSIF tx - start >= PT1 THEN
	Q := FALSE;
	W := TRUE;
	start := tx;
END_IF;

ix := IN_work;
END_FUNCTION_BLOCK

FUNCTION_BLOCK TP_X
VAR_INPUT
	IN : BOOL;
	PT : TIME;
END_VAR
VAR_OUTPUT
	Q : BOOL;
	ET : TIME;
END_VAR
VAR
	edge : BOOL;
	start : TIME;
	tx: TIME;
END_VAR

(* read system_time *)
tx := DWORD_TO_TIME(T_PLC_MS());

(* rising edge trigger *)
IF IN AND NOT edge THEN
	start := tx;
	Q := PT > t#0ms;
ELSIF Q THEN
	ET := tx - start;
	IF ET >= PT THEN
		Q := FALSE;
		ET := t#0ms;
	END_IF;
END_IF;
edge := IN;
END_FUNCTION_BLOCK

FUNCTION_BLOCK FIFO_16
VAR_INPUT
	Din : DWORD;
	E : BOOL := TRUE;
	RD : BOOL;
	WD : BOOL;
	RST : BOOL;
END_VAR
VAR_OUTPUT
	Dout : DWORD;
	EMPTY : BOOL := TRUE;
	FULL : BOOL;
END_VAR
VAR
	fifo : ARRAY[0..n] OF DWORD;
	pr : INT;
	pw : INT;
END_VAR
VAR CONSTANT
	n : INT := 16;	(* changing this value will chage the number of stored elements in the fifo *)
END_VAR

IF RST THEN
	pw := pr;
	FULL := FALSE;
	EMPTY := TRUE;
	Dout := 0;
ELSIF E THEN
	IF NOT EMPTY AND RD THEN
		Dout := fifo[pr];
		pr := INC1(pr,n);
		EMPTY := pr = pw;
		FULL := FALSE;
	END_IF;
	IF NOT FULL AND WD THEN
		fifo[pw] := Din;
		pw := INC1(pw,n);
		FULL := pw = pr;
		EMPTY := FALSE;
	END_IF;
END_IF;
END_FUNCTION_BLOCK

FUNCTION_BLOCK FIFO_32
VAR_INPUT
	Din : DWORD;
	E : BOOL := TRUE;
	RD : BOOL;
	WD : BOOL;
	RST : BOOL;
END_VAR
VAR_OUTPUT
	Dout : DWORD;
	EMPTY : BOOL := TRUE;
	FULL : BOOL;
END_VAR
VAR
	fifo : ARRAY[0..n] OF DWORD;
	pr : INT;
	pw : INT;
END_VAR
VAR CONSTANT
	n : INT := 32;	(* changing this value will chage the number of stored elements in the fifo *)
END_VAR

IF RST THEN
	pw := pr;
	FULL := FALSE;
	EMPTY := TRUE;
	Dout := 0;
ELSIF E THEN
	IF NOT EMPTY AND RD THEN
		Dout := fifo[pr];
		pr := INC1(pr,n);
		EMPTY := pr = pw;
		FULL := FALSE;
	END_IF;
	IF NOT FULL AND WD THEN
		fifo[pw] := Din;
		pw := INC1(pw,n);
		FULL := pw = pr;
		EMPTY := FALSE;
	END_IF;
END_IF;
END_FUNCTION_BLOCK

FUNCTION_BLOCK STACK_16
VAR_INPUT
	Din : DWORD;
	E : BOOL := TRUE;
	RD : BOOL;
	WD : BOOL;
	RST : BOOL;
END_VAR
VAR_OUTPUT
	Dout : DWORD;
	EMPTY : BOOL := TRUE;
	FULL : BOOL;
END_VAR
VAR
	stack : ARRAY[0..n] OF DWORD;
	pt : INT;
END_VAR
VAR CONSTANT
	n : INT := 15;	(* changing this value will chage the number of stored elements in the fifo *)
END_VAR

IF RST THEN
	(* asynchronous reset for the fifo *)
	pt := 0;
	EMPTY := TRUE;
	FULL := FALSE;
	Dout := 0;
ELSIF E THEN
	IF NOT EMPTY AND RD THEN
		(* read one element *)
		pt := pt - 1;
		Dout := stack[pt];
		EMPTY := pt = 0;
		FULL := FALSE;
	END_IF;
	IF NOT FULL AND WD THEN
		(* write one element *)
		stack[pt] := Din;
		pt := pt + 1;
		FULL := pt > n;
		EMPTY := FALSE;
	END_IF;
END_IF;
END_FUNCTION_BLOCK

FUNCTION_BLOCK STACK_32
VAR_INPUT
	Din : DWORD;
	E : BOOL := TRUE;
	RD : BOOL;
	WD : BOOL;
	RST : BOOL;
END_VAR
VAR_OUTPUT
	Dout : DWORD;
	EMPTY : BOOL := TRUE;
	FULL : BOOL;
END_VAR
VAR
	stack : ARRAY[0..n] OF DWORD;
	pt : INT;
END_VAR
VAR CONSTANT
	n : INT := 31;	(* changing this value will chage the number of stored elements in the fifo *)
END_VAR

IF RST THEN
	(* asynchronous reset for the fifo *)
	pt := 0;
	EMPTY := TRUE;
	FULL := FALSE;
	Dout := 0;
ELSIF E THEN
	IF NOT EMPTY AND RD THEN
		(* read one element *)
		pt := pt - 1;
		Dout := stack[pt];
		EMPTY := pt = 0;
		FULL := FALSE;
	END_IF;
	IF NOT FULL AND WD THEN
		(* write one element *)
		stack[pt] := Din;
		pt := pt + 1;
		FULL := pt > n;
		EMPTY := FALSE;
	END_IF;
END_IF;
END_FUNCTION_BLOCK

FUNCTION CRC_GEN : DWORD

VAR_INPUT
	PT : REF_TO ARRAY[0..32000] OF BYTE;
	SIZE : INT;
	PL : INT;
	PN : DWORD;
	INIT : DWORD;
	REV_IN : BOOL;
	REV_OUT : BOOL;
	XOR_OUT : DWORD;
END_VAR
VAR
	pos : INT;
	shift : INT;
	dx: BYTE;
	bits: INT;
	PN_work : DWORD;
END_VAR

(* align polygon *)
shift := 32 - PL;
PN_work := SHL(PN, shift); (* beedance: a copy, as IEC 61131-3 does not let a function assign its input *)

FOR pos := 0 TO 3 DO
	IF REV_IN THEN CRC_GEN := SHL(CRC_GEN, 8) OR REVERSE(PT^[pos]); ELSE CRC_GEN := SHL(CRC_GEN, 8) OR PT^[pos]; END_IF;
END_FOR;
pos := 4;

(* xor with init value *)
CRC_GEN := CRC_GEN XOR SHL(init, shift);

(* calculate CRC for each byte *)
WHILE pos < size DO
	IF REV_IN THEN DX := REVERSE(PT^[pos]); ELSE DX := PT^[pos]; END_IF;
	pos := pos + 1;
	(* crc calculation for one byte *)
	FOR bits := 0 TO 7 DO
		IF CRC_GEN.31 THEN
			CRC_GEN := (SHL(CRC_GEN, 1) OR BOOL_TO_DWORD(DX.7)) XOR PN_work;
		ELSE
			CRC_GEN := SHL(CRC_GEN, 1) OR BOOL_TO_DWORD(DX.7);
		END_IF;
		dx := SHL(dx, 1);
	END_FOR;
END_WHILE;

(* all bytes are processed, need to finish the registers 32 bits *)
FOR bits := 0 TO 31 DO
	IF CRC_GEN.31 THEN
		CRC_GEN := (SHL(CRC_GEN, 1) ) XOR PN_work;
	ELSE
		CRC_GEN := SHL(CRC_GEN, 1);
	END_IF;
END_FOR;

(* final XOR *)
CRC_GEN := SHR(CRC_GEN, shift) XOR XOR_OUT;

(* reverse the crc_out put if necessary *)
IF REV_OUT THEN CRC_GEN := REFLECT(CRC_GEN, PL); END_IF;
END_FUNCTION

FUNCTION_BLOCK MATRIX
VAR_INPUT
	x1, x2, x3, x4, X5 : BOOL;
END_VAR
VAR_INPUT CONSTANT
	Release : BOOL;
END_VAR
VAR_OUTPUT
	code : BYTE;
	TP : BOOL;
	y1: BOOL := TRUE;
	y2, y3, y4 : BOOL;
END_VAR
VAR
	line : BYTE;
	X : ARRAY[0..3] OF BYTE; (* scan line inputs *)
	L : ARRAY[0..3] OF BYTE; (* scan line status *)
	i: INT;
	temp: BYTE;
END_VAR

TP := FALSE;
CODE := 0;
(* read scan lines *)
X[line].0 := X1;
X[line].1 := X2;
X[line].2 := X3;
X[line].3 := X4;
X[line].4 := X5;

(* compare for change *)
FOR i := 0 TO 3 DO
	IF X[i] <> L[i] THEN
		(* scan line information has changed code need to be found and generated *)
		temp := x[i] XOR L[i];
		IF temp.0 THEN
			CODE := 1;
			code.7 := X[i].0;
			L[i].0 := X[i].0;
		ELSIF temp.1 THEN
			code := 2;
			code.7 := X[i].1;
			L[i].1 := X[i].1;
		ELSIF temp.2 THEN
			code := 3;
			code.7 := X[i].2;
			L[i].2 := X[i].2;
		ELSIF temp.3 THEN
			CODE := 4;
			CODE.7 := X[i].3;
			L[i].3 := X[i].3;
		ELSIF temp.4 THEN
			CODE := 5;
			CODE.7 := X[i].4;
			L[i].4 := X[i].4;
		END_IF;
		TP := TRUE;
		CODE.4 := Line.0;
		CODE.5 := Line.1;
		CODE.6 := Line.2;

		(* check if release codes need to be killed *)
		IF NOT release AND CODE < 127 THEN
			CODE := 0;
			TP := FALSE;
		END_IF;
		EXIT;
	END_IF;
END_FOR;

(* increment scan line every cycle *)
line := ULINT_TO_BYTE((BYTE_TO_ULINT(line) + 1) MOD 256) AND 2#0000_0011;
temp := SHL(BYTE#1,line);
Y1 := temp.0;
Y2 := temp.1;
Y3 := temp.2;
Y4 := temp.3;
END_FUNCTION_BLOCK

// Commented out for beedance: it uses CODE, which is commented out.
// FUNCTION_BLOCK PIN_CODE
// VAR_INPUT
// 	CB : BYTE;
// 	E : BOOL;
// END_VAR
// VAR_INPUT CONSTANT
// 	PIN : STRING(8);
// END_VAR
// VAR_OUTPUT
// 	TP : BOOL;
// END_VAR
// VAR
// 	POS: INT := 1;
// END_VAR
//
// tp := FALSE;
// IF e THEN
// 	IF CB = CODE(pin, pos) THEN
// 		pos := pos + 1;
// 		IF pos > LEN(PIN) THEN
// 			(* proper code is detected *)
// 			TP := TRUE;
// 			pos := 1;
// 		END_IF;
// 	ELSE
// 		pos := 1;
// 	END_IF;
// END_IF;
// END_FUNCTION_BLOCK

FUNCTION _ARRAY_ABS : BOOL
VAR_INPUT
	pt : REF_TO ARRAY[0..32000] OF REAL;
	size : UINT;
END_VAR
VAR
	i: UINT;
	stop: UINT;
END_VAR

stop := ((size) / 4)-1;
FOR i := 0 TO stop DO
	PT^[i] := ABS(PT^[i]);
END_FOR;
_ARRAY_ABS := TRUE;
END_FUNCTION

FUNCTION _ARRAY_ADD : BOOL
VAR_INPUT
	pt : REF_TO ARRAY[0..32000] OF REAL;
	size : UINT;
	X : REAL;
END_VAR
VAR
	i: UINT;
	stop: UINT;
END_VAR

stop := ((size) / 4)-1;
FOR i := 0 TO stop DO
	PT^[i] := PT^[i] + X;
END_FOR;
_ARRAY_ADD := TRUE;
END_FUNCTION

FUNCTION _ARRAY_INIT : BOOL
VAR_INPUT
	pt : REF_TO ARRAY[0..32000] OF REAL;
	size : UINT;
	init : REAL;
END_VAR
VAR
	i: UINT;
	stop: UINT;
END_VAR

stop := ((size) / 4)-1;
FOR i := 0 TO stop DO
	pt^[i] := init;
END_FOR;

_array_init := TRUE;
END_FUNCTION

FUNCTION _ARRAY_MEDIAN : REAL
VAR_INPUT
	pt : REF_TO ARRAY[0..32000] OF REAL;
	size : UINT;
END_VAR
VAR
	i: UINT;
	stop: UINT;
END_VAR

_ARRAY_SORT(pt,size);
stop := ((size) / 4)-1;
IF EVEN(UINT_TO_INT(stop)) THEN
	_ARRAY_MEDIAN := pt^[((stop) / 2)];
ELSE
	i := ((stop) / 2);
	_ARRAY_MEDIAN := (pt^[i] + pt^[i+1]) * 0.5;
END_IF;
END_FUNCTION

FUNCTION _ARRAY_MUL : BOOL
VAR_INPUT
	pt : REF_TO ARRAY[0..32000] OF REAL;
	size : UINT;
	X : REAL;
END_VAR
VAR
	i: UINT;
	stop: UINT;
END_VAR

stop := ((size) / 4)-1;
FOR i := 0 TO stop DO
	PT^[i] := PT^[i] * X;
END_FOR;
_ARRAY_MUL := TRUE;
END_FUNCTION

FUNCTION _ARRAY_SHUFFLE : BOOL
VAR_INPUT
	pt : REF_TO ARRAY[0..32000] OF REAL;
	size : UINT;
END_VAR
VAR
	temp : REAL;
	pos  : INT;
	i: INT;
	stop: INT;
END_VAR

stop := UINT_TO_INT(((size) / 4)-1);
FOR i := 0 TO stop DO
        pos := RDM2(i+pos,0,stop);
        (* swap elements *)
        temp := pt^[i];
        pt^[i] := pt^[pos];
        pt^[pos] := temp;
END_FOR;

_ARRAY_SHUFFLE := TRUE;
END_FUNCTION

FUNCTION _ARRAY_SORT : BOOL
VAR_INPUT
	PT : REF_TO ARRAY[1..32000] OF REAL;
	SIZE : UINT;
END_VAR
VAR
	stack_count: UINT;				(* loop variable stack*)
	stack: ARRAY[1..32] OF UINT;	(* stack size ~ 1.6*Log(n)/log(2) *)
										(* stack size 32 => ~1 million elements *)
	links: UINT;						(* first element of the array *)
	rechts: UINT;						(* last element of the array *)
	pivot: REAL;						(* temporary threshold for the swap condition *)
	i: UINT;							(* loop variable 1 *)
	j: UINT;							(* loop variable 2 *)
	ende_innen: BOOL;				(* end of inner loop *)
	ende_aussen: BOOL;				(* end of outer loop *)
	tmp: REAL;						(* helper variable for swapping values *)
END_VAR

(* start values for the array size *)
links := 1;					(* first element of the array *)
rechts := ((size) / 4);		(* last element of the array *)
stack_count := 1;			(* loop variable stack *)

WHILE NOT ende_aussen DO						(* outer loop *)
	IF links < rechts THEN
		pivot := PT^[((rechts+links) / 2)];			(* value of the middle element as pivot value *)
		i := links -1;
		j := rechts +1;

		(* inner loop, partition the array *)
		ende_innen := FALSE;
		REPEAT

			(* ascending order *)
			REPEAT	i := i+1;	UNTIL (PT^[i] >= pivot) OR NOT (i < rechts)	END_REPEAT;
			REPEAT	j := j-1;	UNTIL (PT^[j] <= pivot) OR NOT (j > links)	END_REPEAT;

			(*descending order *)
(*			REPEAT	i := i+1;	UNTIL (PT^[i] <= pivot) OR NOT (i < rechts)	END_REPEAT	*)
(*			REPEAT	j := j-1;	UNTIL (PT^[j] >= pivot) OR NOT (j > links)	END_REPEAT	*)

			IF i >= j THEN
				ende_innen := TRUE;
			ELSE
				   tmp := PT^[j];
				PT^[j] := PT^[i];
				PT^[i] := tmp;
			END_IF;

		UNTIL ende_innen END_REPEAT;

		(* Push stack *)
		stack[stack_count] := rechts;		(* sort the right part later *)
		IF Stack_count < 32 THEN
			stack_count := stack_count +1;
		ELSE
			ende_aussen := TRUE;
			_ARRAY_SORT := FALSE;					(* error: stack too small *)
		END_IF;

		(* sort the left part *)
		rechts := MAX(links, i-1);

	ELSE

		IF stack_count = 1 THEN
			ende_aussen := TRUE;
		ELSE

			links := rechts+1;

			(* pop stack *)
			stack_count := stack_count -1;		(* now sort the right part *)
			rechts:= stack[stack_count];
		END_IF;

	END_IF;

END_WHILE;

_ARRAY_SORT := TRUE;				(* sorting finished *)
END_FUNCTION

FUNCTION ARRAY_AVG : REAL
VAR_INPUT
	pt : REF_TO ARRAY[0..32000] OF REAL;
	size : UINT;
END_VAR
VAR
	i: UINT;
	stop: UINT;
END_VAR

stop := ((size) / 4)-1;
ARRAY_AVG := pt^[0];
FOR i := 1 TO stop DO
	ARRAY_AVG := ARRAY_AVG + pt^[i];
END_FOR;
ARRAY_AVG := ARRAY_AVG / UINT_TO_REAL(stop + 1);
END_FUNCTION

FUNCTION ARRAY_GAV : REAL
VAR_INPUT
	pt : REF_TO ARRAY[0..32000] OF REAL;
	size : UINT;
END_VAR
VAR
	i: UINT;
	stop: UINT;
END_VAR

stop := ((size) / 4)-1;
ARRAY_GAV := 1.0;
FOR i := 0 TO stop DO
	IF pt^[i] > 0.0 THEN
		ARRAY_GAV := ARRAY_GAV * pt^[i];
	ELSE
		ARRAY_GAV := 0.0;
		RETURN;
	END_IF;
END_FOR;
ARRAY_GAV := SQRTN(ARRAY_GAV,UINT_TO_INT(stop)+1);
END_FUNCTION

FUNCTION ARRAY_HAV : REAL
VAR_INPUT
	pt : REF_TO ARRAY[0..32000] OF REAL;
	size : UINT;
END_VAR
VAR
	i: UINT;
	stop: UINT;
END_VAR

stop := ((size) / 4)-1;
FOR i := 0 TO stop DO
	IF pt^[i] <> 0.0 THEN
		ARRAY_HAV := ARRAY_HAV + 1.0 / pt^[i];
	ELSE
		ARRAY_HAV := 0.0;
		RETURN;
	END_IF;
END_FOR;
ARRAY_HAV := UINT_TO_REAL(stop + 1) / ARRAY_HAV;
END_FUNCTION

// Commented out for beedance: it takes SIZEOF(pt), the size of a pointer, as the size of an element; a beedance reference (REF_TO) has no size of its own.
// FUNCTION ARRAY_MAX : REAL
// VAR_INPUT
// 	pt : REF_TO ARRAY[0..32000] OF REAL;
// 	size : UINT;
// END_VAR
// VAR
// 	i: UINT;
// 	stop: UINT;
// END_VAR
//
// stop := (size -SIZEOF(pt)) / SIZEOF(pt);
// array_max := pt^[0];
// FOR i := 1 TO stop DO
// 	IF pt^[i] > array_max THEN array_max := pt^[i]; END_IF;
// END_FOR;
// END_FUNCTION

// Commented out for beedance: it takes SIZEOF(pt), the size of a pointer, as the size of an element; a beedance reference (REF_TO) has no size of its own.
// FUNCTION ARRAY_MIN : REAL
// VAR_INPUT
// 	pt : REF_TO ARRAY[0..32000] OF REAL;
// 	size : UINT;
// END_VAR
// VAR
// 	i: UINT;
// 	stop: UINT;
// END_VAR
//
// stop := (size - SIZEOF(pt)) / SIZEOF(pt);
// array_min := pt^[0];
// FOR i := 1 TO stop DO
// 	IF pt^[i] < array_min THEN array_min := pt^[i]; END_IF;
// END_FOR;
// END_FUNCTION

FUNCTION ARRAY_SDV : REAL
VAR_INPUT
	pt : REF_TO ARRAY[0..32000] OF REAL;
	size : UINT;
END_VAR

(* standard deviation is simply the square root of the variance *)

array_sdv := SQRT(array_var(pt, size));
END_FUNCTION

// Commented out for beedance: it takes SIZEOF(pt), the size of a pointer, as the size of an element; a beedance reference (REF_TO) has no size of its own.
// FUNCTION ARRAY_SPR : REAL
// VAR_INPUT
// 	pt : REF_TO ARRAY[0..32000] OF REAL;
// 	size : UINT;
// END_VAR
// VAR
// 	i: UINT;
// 	stop: UINT;
// 	array_max : REAL;
// 	array_min : REAL;
// END_VAR
//
// stop := (size -SIZEOF(pt)) / SIZEOF(pt);
// array_min := pt^[0];
// array_max := pt^[0];
// FOR i := 1 TO stop DO
// 	IF pt^[i] > array_max THEN array_max := pt^[i];
// 	ELSIF pt^[i] < array_min THEN array_min := pt^[i];
// 	END_IF;
// END_FOR;
// array_spr := array_max - array_min;
// END_FUNCTION

// Commented out for beedance: it takes SIZEOF(pt), the size of a pointer, as the size of an element; a beedance reference (REF_TO) has no size of its own.
// FUNCTION ARRAY_SUM : REAL
// VAR_INPUT
// 	pt : REF_TO ARRAY[0..32000] OF REAL;
// 	size : UINT;
// END_VAR
// VAR
// 	i: UINT;
// 	stop: UINT;
// END_VAR
//
// stop := (size -SIZEOF(pt)) / SIZEOF(pt);
// array_sum := pt^[0];
// FOR i := 1 TO stop DO
// 	array_sum := array_sum + pt^[i];
// END_FOR;
// END_FUNCTION

FUNCTION ARRAY_TREND : REAL
VAR_INPUT
	pt : REF_TO ARRAY[0..32000] OF REAL;
	size : UINT;
END_VAR
VAR
	i: UINT;
	stop: UINT;
	x: REAL;
	stop2: UINT;
END_VAR

stop := ((size) / 4)-1;
stop2 := ((stop) / 2);
FOR i := 0 TO stop2 DO x := x - pt^[i]; END_FOR;
IF EVEN(UINT_TO_INT(stop)) THEN
	FOR i := stop2 TO stop DO X := X + pt^[i]; END_FOR;
ELSE
	FOR i := stop2 + 1 TO stop DO X := X + pt^[i]; END_FOR;
END_IF;
ARRAY_TREND := x / UINT_TO_REAL(stop2 + 1);
END_FUNCTION

FUNCTION ARRAY_VAR : REAL
VAR_INPUT
	pt : REF_TO ARRAY[0..32000] OF REAL;
	size : UINT;
END_VAR
VAR
	avg : REAL;
	i: UINT;
	stop: UINT;
END_VAR

(* at first we calualte the arithmetic average of the array *)

stop := ((size) / 4)-1;
avg := pt^[0];
FOR i := 1 TO stop DO
	avg := avg + pt^[i];
END_FOR;
avg := avg / UINT_TO_REAL(stop + 1);

(* in a second run we calculate the variance of the array *)

array_var := (pt^[0] - avg) * (pt^[0] - avg);
FOR i := 1 TO stop DO
	array_var := array_var + (pt^[i] - avg) * (pt^[i] - avg);
END_FOR;
ARRAY_VAR := ARRAY_VAR / UINT_TO_REAL(stop);
END_FUNCTION

FUNCTION IS_SORTED : BOOL
VAR_INPUT
	pt : REF_TO ARRAY[0..32000] OF REAL;
	size : UINT;
END_VAR
VAR

	stop: INT;
	i: INT;
END_VAR

stop := UINT_TO_INT(((size) / 4)-2);
FOR i := 0 TO stop DO
	IF pt^[i] > pt^[i+1] THEN
		IS_SORTED := FALSE;
		RETURN;
	END_IF;
END_FOR;

IS_SORTED := TRUE;
END_FUNCTION

FUNCTION CABS : REAL
VAR_INPUT
	X : complex;
END_VAR

CABS := HYPOT(x.re, x.im);
END_FUNCTION

FUNCTION CACOS : complex
VAR_INPUT
	X : complex;
END_VAR
VAR
	Y : complex;
END_VAR

y := CACOSH(x);
CACOS.re := y.im;
CACOS.im := -y.re;
END_FUNCTION

FUNCTION CACOSH : complex
VAR_INPUT
	X : complex;
END_VAR
VAR
	Y : complex;
END_VAR

y.re := (X.re - X.im)*(X.re + X.im) - 1.0;
y.im := 2.0 * X.re * X.im;
y    := CSQRT(y);
y.re := y.re + x.re;
y.im := y.im + x.im;
CACOSH  := CLOG(y);
END_FUNCTION

FUNCTION CADD : complex
VAR_INPUT
	X, Y : complex;
END_VAR

CADD.re := x.re + y.re;
CADD.im := x.im + y.im;
END_FUNCTION

FUNCTION CARG : REAL
VAR_INPUT
	X : complex;
END_VAR

CARG := ATAN2(X.im, X.re);
END_FUNCTION

FUNCTION CASIN : complex
VAR_INPUT
	X : complex;
END_VAR
VAR
	Y : complex;
END_VAR

y.re := -x.im;
y.im := x.re;
y := CASINH(y);
CASIN.re := y.im;
CASIN.im := -y.re;
END_FUNCTION

FUNCTION CASINH : complex
VAR_INPUT
	X : complex;
END_VAR
VAR
	Y : complex;
END_VAR

y.re := (X.re - X.im)*(X.re + X.im) + 1.0;
y.im := 2.0 * X.re * X.im;
y    := CSQRT(y);
y.re := y.re + x.re;
y.im := y.im + x.im;
CASINH  := CLOG(y);
END_FUNCTION

FUNCTION CATAN : complex
VAR_INPUT
	X : complex;
END_VAR
VAR
	r2: REAL;
	num, den : REAL;
END_VAR

r2 := x.re * x.re;
den := 1.0 - r2 - x.im * x.im;
CATAN.re := 0.5 * ATAN(2.0 * x.re / den);
num := x.im + 1.0;
num := r2 + num * num;
den := x.im - 1.0;
den := r2 + den * den;
CATAN.im := 0.25 * (LN(num)-LN(den));
END_FUNCTION

FUNCTION CATANH : complex
VAR_INPUT
	X : complex;
END_VAR
VAR
	i2: REAL;
	num, den : REAL;
END_VAR

i2 := x.im * x.im;
num := 1.0 + x.re;
num := i2 + num * num;
den := 1.0 - x.re;
den := i2 + den * den;
CATANH.re := 0.25 * (LN(num) - LN(den));
den := 1 - x.re * x.re - i2;
CATANH.im := 0.5 * ATAN(2.0 * x.im / den);
END_FUNCTION

FUNCTION CCON : complex
VAR_INPUT
	X : complex;
END_VAR

CCON.re := x.re;
CCON.im := -x.im;
END_FUNCTION

FUNCTION CCOS : complex
VAR_INPUT
	X : complex;
END_VAR

CCOS := CCOSH(CSET(-X.im, X.re));
END_FUNCTION

FUNCTION CCOSH : complex
VAR_INPUT
	X : complex;
END_VAR

CCOSH.re := cosH(x.re) * COS(x.im);
CCOSH.im := sinH(x.re) * SIN(x.im);
END_FUNCTION

FUNCTION CDIV : complex
VAR_INPUT
	X, Y : complex;
END_VAR
VAR
	Temp : REAL;
END_VAR

temp := Y.re * Y.re + Y.im * Y.im;
CDIV.re := (X.re * Y.re + X.im * Y.im) / temp;
CDIV.im := (X.im * Y.re - X.re * Y.im) / temp;
END_FUNCTION

FUNCTION CEXP : complex
VAR_INPUT
	X : complex;
END_VAR
VAR
	Temp : REAL;
END_VAR

temp := EXP(X.re);
CEXP.re := temp * COS(X.im);
CEXP.im := temp * SIN(X.im);
END_FUNCTION

FUNCTION CINV : complex
VAR_INPUT
	X : complex;
END_VAR
VAR
	temp : REAL;
END_VAR

temp := X.re * X.re + X.im * X.im;
CINV.re := X.re / temp;
CINV.im := -X.im / temp;
END_FUNCTION

FUNCTION CLOG : complex
VAR_INPUT
	X : complex;
END_VAR

CLOG.re := LN(HYPOT(X.re, X.im));
CLOG.im := ATAN2(X.im, X.re);
END_FUNCTION

FUNCTION CMUL : complex
VAR_INPUT
	X, Y : complex;
END_VAR

CMUL.re := X.re * Y.re - X.im * Y.im;
CMUL.im := X.re * Y.im + X.im * Y.re;
END_FUNCTION

FUNCTION CPOL : complex
VAR_INPUT
	L : REAL;
	A : REAL;
END_VAR

CPOL.re := L * COS(A);
CPOL.im := L * SIN(A);
END_FUNCTION

FUNCTION CPOW : complex
VAR_INPUT
	X : complex;
	Y : Complex;
END_VAR

CPOW := CEXP(CMUL(Y,CLOG(X)));
END_FUNCTION

FUNCTION CSET : complex
VAR_INPUT
	RE : REAL;
	IM : REAL;
END_VAR

CSET.re := RE;
CSET.im := IM;
END_FUNCTION

FUNCTION CSIN : complex
VAR_INPUT
	X : complex;
END_VAR

CSIN.re := cosH(X.im) * SIN(X.re);
CSIN.im := sinH(X.im) * COS(X.re);
END_FUNCTION

FUNCTION CSINH : complex
VAR_INPUT
	X : complex;
END_VAR

CSINH.re := sinH(X.re) * COS(X.im);
CSINH.im := cosH(X.re) * SIN(X.im);
END_FUNCTION

FUNCTION CSQRT : complex
VAR_INPUT
	X : complex;
END_VAR
VAR
	temp : REAL;
END_VAR

temp := HYPOT(x.re, x.im);
CSQRT.re :=  SQRT(0.5 * (temp + x.re));
CSQRT.im :=  sgn(x.im) * SQRT(0.5 * (temp - x.re));
END_FUNCTION

FUNCTION CSUB : complex
VAR_INPUT
	X, Y : complex;
END_VAR

CSUB.re := X.re - Y.re;
CSUB.im := X.im - Y.im;
END_FUNCTION

FUNCTION CTAN : complex
VAR_INPUT
	X : complex;
END_VAR
VAR
	temp : REAL;
	xi2: REAL;
	xr2: REAL;
END_VAR

xi2 := 2.0 * x.im;
xr2 := 2.0 * x.re;
temp := 1.0 / (COS(xr2) + COSH( xi2));
CTAN.re := temp * SIN(xr2);
CTAN.im := temp * SINH(xi2);
END_FUNCTION

FUNCTION CTANH : complex
VAR_INPUT
	X : complex;
END_VAR
VAR
	temp : REAL;
	xi2: REAL;
	xr2: REAL;
END_VAR

xi2 := 2.0 * x.im;
xr2 := 2.0 * x.re;
temp := 1.0 / (COSH(xr2) + COS(xi2));
CTANH.re := temp * SINH(xr2);
CTANH.im := temp * SIN(xi2);
END_FUNCTION

FUNCTION R2_ABS : REAL2
VAR_INPUT
	X : REAL2;
END_VAR

IF X.RX >= 0.0 THEN
	R2_ABS.RX := X.RX;
	R2_ABS.R1 := X.R1;
ELSE
	R2_ABS.RX := -X.RX;
	R2_ABS.R1 := -X.R1;
END_IF;
END_FUNCTION

FUNCTION R2_ADD : REAL2
VAR_INPUT
	X : Real2;
	Y : REAL;
END_VAR
VAR
	temp: REAL;
END_VAR

temp := X.RX;
R2_ADD.RX := Y + X.R1 + X.RX;
R2_ADD.R1 := temp - R2_ADD.RX + Y + X.R1;
END_FUNCTION

FUNCTION R2_ADD2 : REAL2
VAR_INPUT
	X : Real2;
	Y : REAL2;
END_VAR

R2_ADD2.R1 := X.R1 + Y.R1;
R2_ADD2.RX := X.RX + Y.RX;
END_FUNCTION

FUNCTION R2_MUL : REAL2
VAR_INPUT
	X : REAL2;
	Y : REAL;
END_VAR

R2_MUL.RX := X.RX * Y;
R2_MUL.R1 := X.R1 * Y;
END_FUNCTION

FUNCTION R2_SET : REAL2
VAR_INPUT
	X : REAL;
END_VAR

R2_SET.RX := X;
R2_SET.R1 := 0.0;
END_FUNCTION

FUNCTION F_LIN : REAL
VAR_INPUT
	X : REAL;
	A : REAL;
	B : REAL;
END_VAR

F_lin := A * X + B;
END_FUNCTION

FUNCTION F_LIN2 : REAL
VAR_INPUT
	X : REAL;
	X1: REAL;
	Y1 : REAL;
	X2 : REAL;
	Y2 : REAL;
END_VAR

F_LIN2 := (Y2 - Y1) / (X2 - X1) * (X - X1) + Y1;
END_FUNCTION

FUNCTION F_POLY : REAL
VAR_INPUT
	X : REAL;
	C : ARRAY[0..7] OF REAL;
END_VAR
VAR
END_VAR

F_POLY := ((((((( c[7] * x + c[6] ) * x + c[5] ) * x + c[4] ) * x + c[3] ) * x + c[2] ) * x + c[1] ) * x + c[0] ) ;
END_FUNCTION

FUNCTION F_POWER : REAL
VAR_INPUT
	a : REAL;
	x : REAL;
	n : REAL;
END_VAR

F_POWER := a * EXPT(X, N);
END_FUNCTION

FUNCTION F_QUAD : REAL
VAR_INPUT
	X : REAL;
	A : REAL;
	B : REAL;
	C : REAL;
END_VAR

F_QUAD :=  (A * X + B) * X + C;
END_FUNCTION

FUNCTION FRMP_B : BYTE
VAR_INPUT
	START : BYTE;
	DIR : BOOL;
	TD : TIME;
	TR : TIME;
END_VAR
VAR
END_VAR

IF TD < TR THEN
	FRMP_B := MIN(ULINT_TO_BYTE(DWORD_TO_ULINT(SHL(TIME_TO_DWORD(TD), 8)) / TIME_TO_ULINT(TR)), SEL(DIR, START, ULINT_TO_BYTE(255 - BYTE_TO_ULINT(START))));
	IF DIR THEN
		FRMP_B := ULINT_TO_BYTE(BYTE_TO_ULINT(START) + BYTE_TO_ULINT(FRMP_B));
	ELSE
		FRMP_B := ULINT_TO_BYTE(BYTE_TO_ULINT(START) - BYTE_TO_ULINT(FRMP_B));
	END_IF;
ELSE
	FRMP_B := SEL(DIR, 0, 255);
END_IF;
END_FUNCTION

FUNCTION_BLOCK FT_AVG
VAR_INPUT
	IN : REAL;
	E : BOOL := TRUE;
	N : INT := 32;
	RST : BOOL;
END_VAR
VAR_OUTPUT
	AVG : REAL;
END_VAR
VAR
	buff : DELAY;
	i: INT;
	init : BOOL;
END_VAR

(* limit n to a max of 32 because delay can do max 32 cycles *)
buff.N := LIMIT(0, N, 32);

IF NOT init OR rst THEN
	FOR i := 1 TO N DO
		buff(in := in);
	END_FOR;
	avg := in;
	init := TRUE;
ELSIF E THEN
	buff(in := in);
	avg := avg + (in - buff.out ) / INT_TO_REAL(N);
END_IF;
END_FUNCTION_BLOCK

FUNCTION_BLOCK FT_MIN_MAX
VAR_INPUT
	in : REAL;
	rst : BOOL;
END_VAR
VAR_OUTPUT
	mx : REAL;
	mn : REAL;
END_VAR
VAR
	init: BOOL;
END_VAR

IF rst OR NOT init THEN
	mn := in;
	mx := in;
	init := TRUE;
ELSIF in < mn THEN mn := in;
ELSIF in > mx THEN mx := in;
END_IF;
END_FUNCTION_BLOCK

FUNCTION_BLOCK FT_RMP
VAR_INPUT
	Rmp : BOOL := TRUE;
	in : REAL;
	KR : REAL;
	KF : REAL;
END_VAR
VAR_OUTPUT
	out : REAL;
	busy : BOOL;
	UD : BOOL;
END_VAR
VAR
	tx: TIME;
	last: TIME;
	init: BOOL;
END_VAR

(* read system time *)
tx := DWORD_TO_TIME(T_PLC_MS()) - last;

IF NOT init THEN
	init := TRUE;
	last := tx;
	tx := t#0s;
	out := in;
END_IF;
IF NOT rmp THEN
	out := in;
	busy := FALSE;
ELSIF out > in THEN
	(* ramp down *)
	out := out - TIME_TO_REAL(tx) * 0.001 * KF;
	out := MAX(in, out);
ELSIF out < in THEN
	(* ramp up *)
	out := out + TIME_TO_REAL(tx) * 0.001 * KR;
	out := MIN(in, out);
END_IF;

(* set busy and dir flags *)
IF out < in THEN
	busy := TRUE;
	ud := TRUE;
ELSIF out > in THEN
	busy := TRUE;
	ud := FALSE;
ELSE
	busy := FALSE;
END_IF;
last := last + tx;
END_FUNCTION_BLOCK

FUNCTION LINEAR_INT : REAL
VAR_INPUT
	X : REAL;
	XY : ARRAY[1..20,0..1] OF REAL;
	Pts : INT;
END_VAR
VAR
	i : INT;
END_VAR
VAR
	Pts_work : INT;
END_VAR
(* IEC 61131-3 does not let a POU assign to its inputs, so the body works on copies. *)
Pts_work := Pts;

(*make sure n is bound within the array size *)
Pts_work := MIN(Pts_work,20);

(* calculate the linear segement interpolation *)
i := 2;
WHILE (i < Pts_work) AND (XY[i,0] < X) DO
	i := i + 1;
END_WHILE;

(* calculate the output value on the corresponding segment coordinates *)
LINEAR_INT := ((XY[i,1] - XY[i-1,1]) * X - XY[i,1] * XY[i-1,0] + XY[i-1,1] * XY[i,0]) / (XY[i,0] - XY[i-1,0]);
END_FUNCTION

FUNCTION POLYNOM_INT : REAL
VAR_INPUT
	X : REAL;
	XY : ARRAY[1..5,0..1] OF REAL;
	Pts : INT;
END_VAR
VAR
	I, J : INT;
	stop: INT;
END_VAR
VAR
	XY_work : ARRAY [1 .. 5, 0 .. 1] OF REAL;
	Pts_work : INT;
END_VAR
(* IEC 61131-3 does not let a POU assign to its inputs, so the body works on copies. *)
XY_work := XY;
Pts_work := Pts;

(*make sure n is bound within the array size *)
Pts_work := MIN(Pts_work, 5);

FOR i := 1 TO Pts_work DO
	stop := i + 1;
   	FOR j := Pts_work TO stop BY -1 DO
   		XY_work[j,1] := (XY_work[j,1] - XY_work[j-1,1]) / (XY_work[j,0] - XY_work[j-i,0]);
	END_FOR;
END_FOR;

(* this part is the actual calculation *)
POLYNOM_INT := 0.0;
FOR i := Pts_work TO 1 BY -1 DO
       POLYNOM_INT := POLYNOM_INT * (X - XY_work[i,0]) + XY_work[i,1];
END_FOR;
END_FUNCTION

FUNCTION CIRCLE_A : REAL
VAR_INPUT
	rx : REAL;
	ax : REAL;
END_VAR

circle_A := Rx * RX * 8.726646E-3 * Ax;
END_FUNCTION

FUNCTION CIRCLE_C : REAL
VAR_INPUT
	Rx : REAL;
	Ax : REAL;
END_VAR

circle_C := 1.7453293E-2 * Rx * Ax;
END_FUNCTION

FUNCTION CIRCLE_SEG : REAL
VAR_INPUT
	RX : REAL;
	HX : REAL;
END_VAR

IF RX > 0.0 THEN
	CIRCLE_SEG := 2.0 * ACOS(1.0 - LIMIT(0.0, HX / RX, 2.0));
	CIRCLE_SEG := (CIRCLE_SEG - SIN(CIRCLE_SEG)) *RX * RX / 2.0;
END_IF;
END_FUNCTION

FUNCTION CONE_V : REAL
VAR_INPUT
	rx : REAL;
	hx : REAL;
END_VAR

cone_V := 1.047197551 * RX * RX * hx;
END_FUNCTION

FUNCTION ELLIPSE_A : REAL
VAR_INPUT
	R1 : REAL;
	R2 : REAL;
END_VAR

ELLIPSE_A := math.PI * R1 * R2;
END_FUNCTION

FUNCTION ELLIPSE_C : REAL
VAR_INPUT
	R1 : REAL;
	R2 : REAL;
END_VAR

ELLIPSE_C := math.PI * (3.0 * (R1+R2) - SQRT((3.0 * r1 + R2) * (3.0 * r2 + r1)));
END_FUNCTION

FUNCTION SPHERE_V : REAL
VAR_INPUT
	rx : REAL;
END_VAR

sphere_V := 4.188790205 * Rx * RX * RX;
END_FUNCTION

FUNCTION TRIANGLE_A : REAL
VAR_INPUT
	S1 : REAL;
	A : REAL;
	S2 : REAL;
	S3 : REAL;
END_VAR

IF A = 0.0 THEN
	TRIANGLE_A := SQRT((s1+s2+S3) * (s1+s2-S3) * (S2+S3-S1) * (S3+S1-S2)) * 0.25;
ELSE
	TRIANGLE_A := S1 * S2 * SIN(RAD(A)) * 0.5;
END_IF;
END_FUNCTION

FUNCTION V3_ABS : REAL
VAR_INPUT
	A : Vector_3;
END_VAR

V3_ABS := SQRT(A.X * A.X + A.Y * A.Y + A.Z * A.Z);
END_FUNCTION

FUNCTION V3_ADD : vector_3
VAR_INPUT
	A : Vector_3;
	B : Vector_3;
END_VAR

V3_ADD.X := A.X + B.X;
V3_ADD.Y := A.Y + B.Y;
V3_ADD.Z := A.Z + B.Z;
END_FUNCTION

FUNCTION V3_ANG : REAL
VAR_INPUT
	A : Vector_3;
	B : Vector_3;
END_VAR
VAR
	d : REAL;
END_VAR

d := V3_ABS(A) * V3_ABS(B);
IF d > 0 THEN
	V3_ANG := ACOS(LIMIT(-1.0, V3_DPRO(A, B) / d,1.0));
END_IF;
END_FUNCTION

FUNCTION V3_DPRO : REAL
VAR_INPUT
	A : Vector_3;
	B : Vector_3;
END_VAR

V3_DPRO := A.X * B.X + A.Y * B.Y + A.Z * B.Z;
END_FUNCTION

FUNCTION V3_NORM : vector_3
VAR_INPUT
	A : Vector_3;
END_VAR
VAR
	la: REAL;
END_VAR

la := V3_ABS(A);
IF la > 0.0 THEN
	V3_NORM := V3_SMUL(A, 1.0 / la);
END_IF;
END_FUNCTION

FUNCTION V3_NUL : BOOL
VAR_INPUT
	A : Vector_3;
END_VAR

V3_NUL := A.X = 0.0 AND A.Y = 0.0 AND A.Z = 0.0;
END_FUNCTION

FUNCTION V3_PAR : BOOL
VAR_INPUT
	A : Vector_3;
	B : Vector_3;
END_VAR

V3_PAR := V3_ABS(V3_XPRO(A, B)) = 0.0;
END_FUNCTION

FUNCTION V3_REV : vector_3
VAR_INPUT
	A : Vector_3;
END_VAR

V3_REV.X := -A.X;
V3_REV.Y := -A.Y;
V3_REV.Z := -A.Z;
END_FUNCTION

FUNCTION V3_SMUL : vector_3
VAR_INPUT
	A : Vector_3;
	M : REAL;
END_VAR

V3_SMUL.X := A.X * M;
V3_SMUL.Y := A.Y * M;
V3_SMUL.Z := A.Z * M;
END_FUNCTION

FUNCTION V3_SUB : vector_3
VAR_INPUT
	A : Vector_3;
	B : Vector_3;
END_VAR

V3_SUB.X := A.X - B.X;
V3_SUB.Y := A.Y - B.Y;
V3_SUB.Z := A.Z - B.Z;
END_FUNCTION

FUNCTION V3_XANG : REAL
VAR_INPUT
	A : Vector_3;
END_VAR
VAR
	la: REAL;
END_VAR

la := V3_ABS(a);
IF la > 0.0 THEN
	V3_XANG := ACOS(A.X / la);
END_IF;
END_FUNCTION

FUNCTION V3_XPRO : vector_3
VAR_INPUT
	A : Vector_3;
	B : Vector_3;
END_VAR

V3_XPRO.X := A.Y * B.Z - A.Z * B.Y;
V3_XPRO.Y := A.Z * B.X - A.X * B.Z;
V3_XPRO.Z := A.X * B.Y - A.Y * B.X;
END_FUNCTION

FUNCTION V3_YANG : REAL
VAR_INPUT
	A : Vector_3;
END_VAR
VAR
	la: REAL;
END_VAR

la := V3_ABS(a);
IF la > 0.0 THEN
	V3_YANG := ACOS(A.Y / la);
END_IF;
END_FUNCTION

FUNCTION V3_ZANG : REAL
VAR_INPUT
	A : Vector_3;
END_VAR
VAR
	la: REAL;
END_VAR

la := V3_ABS(a);
IF la > 0.0 THEN
	V3_ZANG := ACOS(A.Z / la);
END_IF;
END_FUNCTION

FUNCTION ACOSH : REAL
VAR_INPUT
	X : REAL;
END_VAR

ACOSH := LN(SQRT(X * X - 1.0) + X);
END_FUNCTION

FUNCTION ACOTH : REAL
VAR_INPUT
	X : REAL;
END_VAR

ACOTH := LN((x+1.0)/(x-1.0))*0.5;
END_FUNCTION

FUNCTION AGDF : REAL
VAR_INPUT
	X : REAL;
END_VAR

AGDF := LN((1.0 + SIN(X)) / COS(X));
END_FUNCTION

FUNCTION ASINH : REAL
VAR_INPUT
	X : REAL;
END_VAR

ASINH := LN(SQRT(X * X + 1.0)+X);
END_FUNCTION

FUNCTION ATAN2 : REAL
VAR_INPUT
	Y : REAL;
	X : REAL;
END_VAR

IF X > 0.0 THEN
	ATAN2 := ATAN(Y/X);
ELSIF X < 0.0 THEN
	IF Y >=0.0 THEN
		ATAN2 := ATAN(Y/X) + MATH.PI;
	ELSE
		ATAN2 := ATAN(Y/X) - MATH.PI;
	END_IF;
ELSIF Y > 0.0 THEN
	ATAN2 := MATH.PI05;
ELSIF Y < 0.0 THEN
	ATAN2 := -MATH.PI05;
ELSE
	ATAN2 := 0.0;
END_IF;
END_FUNCTION

FUNCTION ATANH : REAL
VAR_INPUT
	X : REAL;
END_VAR

ATANH := LN((1.0 + x)/(1.0 - x)) * 0.5;
END_FUNCTION

FUNCTION BETA : REAL
VAR_INPUT
	X : REAL;
	Y : REAL;
END_VAR

BETA := GAMMA(X) * GAMMA(Y) / GAMMA(x + y);
END_FUNCTION

FUNCTION BINOM : DINT
VAR_INPUT
	N : INT;
	K : INT;
END_VAR

VAR
	i: INT;
END_VAR
VAR
	N_work : INT;
	K_work : INT;
END_VAR
(* IEC 61131-3 does not let a POU assign to its inputs, so the body works on copies. *)
N_work := N;
K_work := K;

IF 2 * K_work > N_work THEN
	K_work := N_work - K_work;
END_IF;
IF K_work > N_work THEN
	RETURN;
ELSIF K_work = 0 OR K_work = N_work THEN
	BINOM := 1;
ELSIF K_work = 1 THEN
	BINOM := N_work;
ELSE
	BINOM := N_work;
	N_work := N_work + 1;
	FOR i := 2 TO K_work DO
		BINOM := BINOM * (N_work - i) / i;
	END_FOR;
END_IF;
END_FUNCTION

FUNCTION CAUCHY : REAL
VAR_INPUT
	X : REAL;
	T : REAL;
	U : REAL;
END_VAR
VAR
	tmp: REAL;
END_VAR

tmp := x - t;
CAUCHY := math.PI_INV * U / (U*U + tmp*tmp);
END_FUNCTION

FUNCTION CAUCHYCD : REAL
VAR_INPUT
	X : REAL;
	T : REAL;
	U : REAL;
END_VAR

CAUCHYCD := 0.5 + math.PI_INV * ATAN((X - T) / U);
END_FUNCTION

FUNCTION CEIL : INT
VAR_INPUT
	X : REAL;
END_VAR

CEIL := REAL_TO_INT(x);
IF CEIL < X THEN
	CEIL := CEIL + 1;
END_IF;
END_FUNCTION

FUNCTION CEIL2 : DINT
VAR_INPUT
	X : REAL;
END_VAR

CEIL2 := REAL_TO_DINT(X);
IF DINT_TO_REAL(CEIL2) < X THEN
	CEIL2 := CEIL2 + 1;
END_IF;
END_FUNCTION

FUNCTION CMP : BOOL
VAR_INPUT
	X,Y : REAL;
	N : INT;
END_VAR
VAR
	tmp : REAL;
END_VAR

tmp := ABS(x);
IF tmp > 0.0 THEN
	tmp := EXP10(INT_TO_REAL(FLOOR(LOG(tmp))-N+1));
ELSE
	tmp := EXP10(tmp);
END_IF;
CMP := ABS(X - Y) < tmp;
END_FUNCTION

FUNCTION COSH : REAL
VAR_INPUT
	X : REAL;
END_VAR
VAR
	t: REAL;
END_VAR

T := EXP(X);
COSH := (1.0 / T + T) * 0.5;
END_FUNCTION

FUNCTION COTH : REAL
VAR_INPUT
	X : REAL;
END_VAR

IF X > 20.0 THEN
	COTH :=1.0;
ELSIF X < -20.0 THEN
	COTH := -1.0;
ELSE
	COTH := 1.0 + 2.0 / (EXP(X * 2.0) - 1.0);
END_IF;
END_FUNCTION

FUNCTION D_TRUNC : DINT
VAR_INPUT
	X : REAL;
END_VAR

D_TRUNC := REAL_TO_DINT(X);
IF X > 0.0 THEN
	IF DINT_TO_REAL(D_TRUNC) > X THEN D_TRUNC := D_TRUNC - 1; END_IF;
ELSE
	IF DINT_TO_REAL(D_TRUNC) < X THEN D_TRUNC := D_TRUNC + 1; END_IF;
END_IF;

(* for systems that support a dint truncation this routine can be replaced by trunc() *)
END_FUNCTION

FUNCTION DEC1 : INT
VAR_INPUT
	X : INT;
	N : INT;
END_VAR

IF X = 0 THEN
	DEC1 := N - 1;
ELSE
	DEC1 := X - 1;
END_IF;
END_FUNCTION

FUNCTION DEG : REAL
VAR_INPUT
	rad : REAL;
END_VAR

DEG := MODR(57.29577951308232 * RAD, 360.0);
END_FUNCTION

FUNCTION DIFFER : BOOL
VAR_INPUT
	in1 : REAL;
	in2 : REAL;
	X : REAL;
END_VAR

DIFFER := ABS(in1 - in2) > X;
END_FUNCTION

FUNCTION ERF : REAL
VAR_INPUT
	X : REAL;
END_VAR
VAR
	x2 : REAL;
	ax2 : REAL;
END_VAR

x2 := X*X;
ax2 := 0.147 * x2 + 1.0;
ERF := SQRT(1.0 - EXP(-X2 * ((0.27323954473516 + aX2)/(ax2)))) * SGN(x);
END_FUNCTION

FUNCTION ERFC : REAL
VAR_INPUT
	X : REAL;
END_VAR

ERFC := 1.0 - ERF(X);
END_FUNCTION

FUNCTION EVEN : BOOL
VAR_INPUT
	in : DINT;
END_VAR

EVEN := NOT in.0;
END_FUNCTION

FUNCTION EXP10 : REAL
VAR_INPUT
	X : REAL;
END_VAR

EXP10 := EXP(X * 2.30258509299405);
END_FUNCTION

FUNCTION EXPN : REAL
VAR_INPUT
	X : REAL;
	N : INT;
END_VAR
VAR
	sign: BOOL;
END_VAR
VAR
	X_work : REAL;
	N_work : INT;
END_VAR
(* IEC 61131-3 does not let a POU assign to its inputs, so the body works on copies. *)
X_work := X;
N_work := N;

sign := N_work.15;
N_work := ABS(N_work);
IF N_work.0 THEN EXPN := X_work; ELSE EXPN := 1.0; END_IF;
N_work := N_work / 2;
WHILE N_work > 0 DO
   X_work := X_work * X_work;
   IF N_work.0 THEN EXPN := EXPN * X_work; END_IF;
   N_work := N_work / 2;
END_WHILE;
IF sign THEN EXPN := 1.0 / EXPN; END_IF;
END_FUNCTION

FUNCTION FACT : DINT
VAR_INPUT
	X : INT;
END_VAR

IF X >= 0 AND X <= 12 THEN
	FACT := math.FACTS[X];
ELSE
	FACT := -1;
END_IF;
END_FUNCTION

FUNCTION FIB : DINT
VAR_INPUT
	X : INT;
END_VAR
VAR
	t1, t2: DINT;
END_VAR
VAR
	X_work : INT;
END_VAR
(* IEC 61131-3 does not let a POU assign to its inputs, so the body works on copies. *)
X_work := X;

IF X_work < 0 OR X_work > 46 THEN
	FIB := -1;
ELSIF X_work < 2 THEN
	FIB := X_work;
	RETURN;
ELSE
	(* the fibonacci number is the sum of the two suceeding fibonaci numbers *)
	(* we store the numbers alternatively in t1 and t2 depending on pt *)
	t2 := 1;
	WHILE X_work > 3 DO
		X_work := X_work-2;
		t1 := t1 + t2;
		t2 := t1 + t2;
	END_WHILE;
	IF X_work > 2 THEN t1 := t1 + t2; END_IF;
	fib := t1 + t2;
END_IF;
END_FUNCTION

FUNCTION FLOOR : INT
VAR_INPUT
	X : REAL;
END_VAR

FLOOR := REAL_TO_INT(X);
IF FLOOR > X THEN
	FLOOR := FLOOR - 1;
END_IF;
END_FUNCTION

FUNCTION FLOOR2 : DINT
VAR_INPUT
	X : REAL;
END_VAR

FLOOR2 := REAL_TO_DINT(X);
IF DINT_TO_REAL(FLOOR2) > X THEN
	FLOOR2 := FLOOR2 - 1;
END_IF;
END_FUNCTION

FUNCTION FRACT : REAL
VAR_INPUT
	x : REAL;
END_VAR

IF ABS(x) < 2.0E9 THEN
	FRACT := x - DINT_TO_REAL(D_TRUNC(x));
ELSE
	FRACT := 0.0;
END_IF;
END_FUNCTION

FUNCTION GAMMA : REAL
VAR_INPUT
	X : REAL;
END_VAR

IF x > 0.0 THEN
	GAMMA := SQRT(math.PI2 / X) * EXPT(math.E_INV * (x + 1.0 / (12.0 * x - 0.1 / X)), X);
END_IF;
END_FUNCTION

FUNCTION GAUSS : REAL
VAR_INPUT
	X : REAL;
	U : REAL;
	SI: REAL;
END_VAR
VAR
	temp: REAL;
	si_inv: REAL;
END_VAR

temp := X - U;
si_inv := 1.0  / si;
GAUSS := EXP(Temp * Temp * si_inv * si_inv * - 0.5) * 0.39894228 * si_inv;
END_FUNCTION

FUNCTION GAUSSCD : REAL
VAR_INPUT
	X : REAL;
	U : REAL;
	SI: REAL;
END_VAR

GAUSSCD := (ERF((X - U) / (SI * 1.414213562)) + 1.0) * 0.5;
END_FUNCTION

FUNCTION GCD : INT
VAR_INPUT
	A : DINT;
	B : DINT;
END_VAR
VAR
	t: DINT;
END_VAR
VAR
	A_work : DINT;
	B_work : DINT;
END_VAR
(* IEC 61131-3 does not let a POU assign to its inputs, so the body works on copies. *)
A_work := A;
B_work := B;

IF A_work = 0 THEN
	GCD := DINT_TO_INT(ABS(B_work));
ELSIF B_work = 0 THEN
	GCD := DINT_TO_INT(ABS(A_work));
ELSE
	A_work := ABS(A_work);
	B_work := ABS(B_work);
	GCD := 1;
	WHILE NOT(A_work.0 OR B_work.0) DO
		A_work := A_work / 2;
		B_work := B_work / 2;
		GCD := GCD * 2;
	END_WHILE;
	WHILE A_work > 0 DO
		IF NOT(A_work.0) THEN A_work := A_work / 2;
		ELSIF NOT(B_work.0) THEN B_work := B_work / 2;
		ELSE
			t:= ABS(A_work-B_work) / 2;
			IF A_work < B_work THEN B_work := t; ELSE A_work := T; END_IF;
		END_IF;
	END_WHILE;
	GCD := GCD * DINT_TO_INT(B_work);
END_IF;
END_FUNCTION

FUNCTION GDF : REAL
VAR_INPUT
	X : REAL;
END_VAR

IF X = 0.0 THEN
	GDF := 0.0;
ELSIF X > 15.0 THEN
	GDF := math.PI05;
ELSIF X < -15.0 THEN
	GDF := -math.PI05;
ELSE
	GDF := ATAN(EXP(X)) * 2.0 - math.PI05;
END_IF;
END_FUNCTION

FUNCTION GOLD : REAL
VAR_INPUT
	X : REAL;
END_VAR

GOLD := (X + SQRT(X*X + 4.0)) * 0.5;
END_FUNCTION

FUNCTION HYPOT : REAL
VAR_INPUT
	X : REAL;
	Y : REAL;
END_VAR

HYPOT := SQRT(x*x + y*y);
END_FUNCTION

FUNCTION INC : INT
VAR_INPUT
	X : INT;
	D : INT;
	M : INT;
END_VAR

IF M + 1 > 0 THEN (* OSCAT 3.36: no MOD 0 *)
	INC := (X + D + M + 1) MOD (M + 1);
ELSE
	INC := 0;
END_IF;
END_FUNCTION

FUNCTION INC1 : INT
VAR_INPUT
	X : INT;
	N : INT;
END_VAR

IF X >= N - 1 THEN
	INC1 := 0;
ELSE
	INC1 := X + 1;
END_IF;
END_FUNCTION

FUNCTION INC2 : INT
VAR_INPUT
	X : INT;
	D : INT;
	L : INT;
	U : INT;
END_VAR
VAR
	tmp: INT;
END_VAR

tmp := U - L + 1;
IF tmp <> 0 THEN (* OSCAT 3.36: no MOD 0 *)
	INC2 := (X + D - L + tmp) MOD tmp + L;
ELSE
	INC2 := L;
END_IF;
END_FUNCTION

FUNCTION INV : REAL
VAR_INPUT
	X : REAL;
END_VAR

IF X <> 0.0 THEN INV := 1.0 / X; END_IF;
END_FUNCTION

// Commented out for beedance: it uses REAL_TO_DW, which is commented out.
// FUNCTION LAMBERT_W : REAL
// VAR_INPUT
// 	X : REAL;
// END_VAR
// VAR
// 	w : REAL;
// 	i : INT;
// 	we: REAL;
// 	w1e: REAL;
// 	last: DWORD;
// 	ewx: REAL;
// END_VAR
//
// (* check for valid input and return -1000 if too low *)
// IF x < -0.367879441171442 THEN
// 	LAMBERT_W := -1000.0;
// 	RETURN;
// (* return 0 if x = 0 *)
// ELSIF x = 0.0 THEN
// 	RETURN;
// (* first an estimate is calculated *)
// ELSIF x <= 500.0 THEN
// 	w := LN(x + 1.0);
// 	w := 0.665 * (1.0 + 0.0195 * w) * w + 0.04;
// ELSE
// 	w := LN(x - 4.0) - (1.0 - 1.0/LN(x)) * LN(LN(x));
// END_IF;
// (* use estimate to calculate exact result *)
// FOR i := 0 TO 5 DO
// 	ewx := EXP(w);
// 	we := w * ewx - x;
// 	w1e := (w+1.0) * ewx;
// 	last := REAL_TO_DW(w) AND 16#FFFF_FFFC;
// 	w := w - (we / (w1e - (w+2.0) * we / (2.0 * w + 2.0)));
// 	IF (REAL_TO_DW(w) AND 16#FFFF_FFFC) = last THEN EXIT; END_IF;
// END_FOR;
// LAMBERT_W := w;
// END_FUNCTION

FUNCTION LANGEVIN : REAL
VAR_INPUT
	X : REAL;
END_VAR

IF X = 0.0 THEN
	LANGEVIN := 0.0;
ELSE
	LANGEVIN := COTH(X) - 1.0 / X;
END_IF;
END_FUNCTION

FUNCTION MAX3 : REAL
VAR_INPUT
	in1 : REAL;
	in2 : REAL;
	in3 : REAL;
END_VAR

MAX3 := MAX(MAX(IN1,IN2),IN3);
END_FUNCTION

FUNCTION MID3 : REAL
VAR_INPUT
	IN1 : REAL;
	IN2 : REAL;
	IN3 : REAL;
END_VAR
VAR
	IN1_work : REAL;
	IN2_work : REAL;
END_VAR
(* IEC 61131-3 does not let a POU assign to its inputs, so the body works on copies. *)
IN1_work := IN1;
IN2_work := IN2;

IF IN1_work > IN2_work THEN MID3 := IN1_work; IN1_work := IN2_work; IN2_work := MID3; END_IF;
IF IN2_work > IN3 THEN IN2_work := IN3; END_IF;
MID3 := SEL(IN1_work > IN2_work, IN2_work, IN1_work);
END_FUNCTION

FUNCTION MIN3 : REAL
VAR_INPUT
	in1 : REAL;
	in2 : REAL;
	in3 : REAL;
END_VAR

MIN3 := MIN(MIN(IN1,IN2),IN3);
END_FUNCTION

FUNCTION MODR : REAL
VAR_INPUT
	IN : REAL;
	DIVI : REAL;
END_VAR

IF divi = 0.0 THEN
	MODR := 0.0;
ELSE
	MODR := in - DINT_TO_REAL(FLOOR2(in / divi)) * divi;
END_IF;
END_FUNCTION

FUNCTION MUL_ADD : REAL
VAR_INPUT
	X : REAL;
	K : REAL;
	O : REAL;
END_VAR

MUL_ADD := X * K + O;
END_FUNCTION

FUNCTION NEGX : REAL
VAR_INPUT
	X : REAL;
END_VAR

NEGX := -X;
END_FUNCTION

FUNCTION RAD : REAL
VAR_INPUT
	DEG : REAL;
END_VAR

RAD := MODR(0.0174532925199433 * DEG, math.PI2);
END_FUNCTION

FUNCTION RDM : REAL
VAR_INPUT
	last : REAL;
END_VAR
VAR
	tn : DWORD;
	tc : INT;
END_VAR

tn := T_PLC_MS();
tc := BIT_COUNT(tn);
tn.31 := tn.2;
tn.30 := tn.5;
tn.29 := tn.4;
tn.28 := tn.1;
tn.27 := tn.0;
tn.26 := tn.7;
tn.25 := tn.6;
tn.24 := tn.3;
tn := ROL(tn,BIT_COUNT(tn)) OR 16#80000001;
tn := ULINT_TO_DWORD(DWORD_TO_ULINT(tn) MOD 71474513 + INT_TO_ULINT(tc + 77));
RDM := FRACT(DWORD_TO_REAL(tn) / 10000000.0 * (math.E - LIMIT(0.0,last,1.0)));
END_FUNCTION

FUNCTION RDM2 : INT
VAR_INPUT
	last : INT;
	low : INT;
	high : INT;
END_VAR

RDM2 := TRUNC(RDM(FRACT(last * math.PI)) * (high - low + 1)) + low;
END_FUNCTION

FUNCTION RDMDW : DWORD
VAR_INPUT
	last : DWORD;
END_VAR
VAR
	RX: REAL;
	M: REAL;
END_VAR

M := BIT_COUNT(last);
RX := RDM(FRACT(M * math.PI));
RDMDW := SHL(REAL_TO_DWORD(rx*65535),16);
RX := RDM(FRACT(M * math.E));
RDMDW := RDMDW OR (REAL_TO_DWORD(rx*65535) AND 16#0000FFFF);
END_FUNCTION

FUNCTION REAL_TO_FRAC : FRACTION
VAR_INPUT
	X : REAL;					(* value to be converted into a fraction *)
	N : INT;					(* maximum size of the denominator *)
END_VAR
VAR
	temp : DINT;				(* flag for calculations *)

	sign: BOOL;					(* sign of the input value *)
	X_gerundet: DINT;			(* value of fraction, rounded to an integer *)
	X_ohne_Nachkomma: REAL;		(* value of fraction, without decimal places *)
	Numerator:       DINT := 1;	(* initial value numerator  *)
	Denominator:     DINT := 0;	(* initial value denominator *)
	Numerator_old:   DINT := 0;	(* initial value numerator of the last calculation  *)
	Denominator_old: DINT := 1;	(* initial value numerator of the last calculation   *)

END_VAR
VAR
	X_work : REAL;
END_VAR
(* IEC 61131-3 does not let a POU assign to its inputs, so the body works on copies. *)
X_work := X;

IF X_work < 0.0 THEN
	sign := TRUE;								(* remember sign *)
	X_work := ABS(X_work);								(* calculate absolute value *)
END_IF;

REPEAT
	X_gerundet := REAL_TO_DINT(X_work);

	(* calculate numerator *)
	temp := numerator * X_gerundet + numerator_old;		(* extend numerator by the integer part *)
	numerator_old := numerator;							(* store numerator of the last calculation *)
	numerator := temp;									(* store numerator of this calculation *)

	(* calculate denominator *)
	temp := denominator * X_gerundet + denominator_old;	(* extend denominator by the integer part *)
	denominator_old := denominator;						(* store denominator of the last calculation *)
	denominator := temp;								(* store denominator of this calculation *)

	(* calculate remainder *)
	X_ohne_Nachkomma := DINT_TO_REAL(X_gerundet);
	IF X_work = X_ohne_Nachkomma THEN						(* fraction divides without remainder *)
		IF ABS(denominator) <= N THEN						(* no rounding error *)
			numerator_old := numerator;					(* Numerator_old is returned by the function *)
			denominator_old := denominator;			(* Denominator_old is returned by the function *)
		END_IF
		EXIT;											(* no further calculation necessary *)
	ELSE
		X_work := 1.0 / (X_work - X_ohne_Nachkomma);				(* reciprocal of the remainder -> new fraction *)
	END_IF

UNTIL
	ABS(Denominator) > N
END_REPEAT

(* correct sign if X was negative *)
IF sign THEN
	REAL_TO_FRAC.NUMERATOR := -1 * ABS(DINT_TO_INT(numerator_old));
ELSE
	REAL_TO_FRAC.NUMERATOR :=  ABS(DINT_TO_INT(numerator_old));
END_IF
REAL_TO_FRAC.DENOMINATOR := ABS(DINT_TO_INT(denominator_old));
END_FUNCTION

FUNCTION RND : REAL
VAR_INPUT
	X : REAL;
	N : INT;
END_VAR
VAR
	M : REAL;
END_VAR

IF X = 0.0 THEN
	RND := 0.0;
ELSE
	M := EXPN(10.0,N - CEIL(LOG(ABS(X))));
	RND := DINT_TO_REAL(REAL_TO_DINT(X * M)) / M;
END_IF;
END_FUNCTION

FUNCTION ROUND : REAL
VAR_INPUT
	in : REAL;
	N : INT;
END_VAR
VAR
	X: REAL;
END_VAR

X := setup.DECADES[LIMIT(0,N,8)];
ROUND := DINT_TO_REAL(REAL_TO_DINT(in * X)) / X;
END_FUNCTION

FUNCTION SGN : INT
VAR_INPUT
	X : REAL;
END_VAR

IF X > 0 THEN
	SGN := 1;
ELSIF X < 0 THEN
	SGN := -1;
ELSE
	SGN := 0;
END_IF;
END_FUNCTION

FUNCTION SIGMOID : REAL
VAR_INPUT
	X : REAL;
END_VAR

IF X > 20.0 THEN
	SIGMOID := 1.0;
ELSIF x < -85.0 THEN
	SIGMOID := 0.0;
ELSE
	SIGMOID := 1.0 / (1.0 + EXP(-X));
END_IF;
END_FUNCTION

FUNCTION SIGN_I : BOOL
VAR_INPUT
	IN : DINT;
END_VAR

SIGN_I := in.31;
END_FUNCTION

FUNCTION SIGN_R : BOOL
VAR_INPUT
	in : REAL;
END_VAR

SIGN_R := in < 0.0;
END_FUNCTION

FUNCTION SINC : REAL
VAR_INPUT
	X : REAL;
END_VAR

IF X = 0.0 THEN
	SINC := 1.0;
ELSE
	SINC := SIN(x) / x;
END_IF;
END_FUNCTION

FUNCTION SINH : REAL
VAR_INPUT
	X : REAL;
END_VAR

IF ABS(x) < 2E-3 THEN
	SINH := X;
ELSE
	SINH := (EXP(x) - EXP(-x)) * 0.5;
END_IF;
END_FUNCTION

FUNCTION SQRTN : REAL
VAR_INPUT
	X : REAL;
	N : INT;
END_VAR

IF N > 0 THEN
	SQRTN := EXP(LN(x) / INT_TO_REAL(n));
ELSE
	SQRTN := 0.0;
END_IF;
END_FUNCTION

FUNCTION TANC : REAL
VAR_INPUT
	X : REAL;
END_VAR

IF X = 0.0 THEN
	TANC := 1.0;
ELSE
	TANC := TAN(x) / x;
END_IF;
END_FUNCTION

FUNCTION TANH : REAL
VAR_INPUT
	X : REAL;
END_VAR

IF X > 20.0 THEN
	TANH := 1.0;
ELSIF X < -20.0 THEN
	TANH := -1.0;
ELSE
	TANH := 1.0 - 2.0 / (EXP(2.0 * x) + 1.0);
END_IF;
END_FUNCTION

FUNCTION WINDOW : BOOL
VAR_INPUT
	low : REAL;
	in : REAL;
	high : REAL;
END_VAR

WINDOW := in < high AND in > low;
END_FUNCTION

FUNCTION WINDOW2 : BOOL
VAR_INPUT
	LOW : REAL;
	IN : REAL;
	HIGH : REAL;
END_VAR

WINDOW2 := IN >= LOW AND IN <= HIGH;
END_FUNCTION

FUNCTION_BLOCK ESR_COLLECT
VAR_INPUT
	ESR_0, ESR_1, ESR_2, ESR_3, ESR_4, ESR_5, ESR_6, ESR_7 : ARRAY [0..3] OF esr_data;
	rst : BOOL;
END_VAR
VAR_IN_OUT
	pos : INT;
END_VAR
VAR_OUTPUT
	ESR_OUT : ARRAY[0..31] OF esr_data;
END_VAR
VAR CONSTANT
	max_in : INT := 3; (* max limit of input array *)
	max_out : INT := 32; (* number of elements in array *)
END_VAR
VAR
	cnt : INT := -1;
END_VAR

IF rst OR cnt < 0 THEN
	pos := -1;
ELSE
	FOR cnt := 0 TO max_in DO
	IF esr_0[cnt].typ > 0 THEN pos := INC1(pos, max_out); esr_out[pos] := esr_0[cnt]; END_IF;
	IF esr_1[cnt].typ > 0 THEN pos := INC1(pos, max_out); esr_out[pos] := esr_1[cnt]; END_IF;
	IF esr_2[cnt].typ > 0 THEN pos := INC1(pos, max_out); esr_out[pos] := esr_2[cnt]; END_IF;
	IF esr_3[cnt].typ > 0 THEN pos := INC1(pos, max_out); esr_out[pos] := esr_3[cnt]; END_IF;
	IF esr_4[cnt].typ > 0 THEN pos := INC1(pos, max_out); esr_out[pos] := esr_4[cnt]; END_IF;
	IF esr_5[cnt].typ > 0 THEN pos := INC1(pos, max_out); esr_out[pos] := esr_5[cnt]; END_IF;
	IF esr_6[cnt].typ > 0 THEN pos := INC1(pos, max_out); esr_out[pos] := esr_6[cnt]; END_IF;
	IF esr_7[cnt].typ > 0 THEN pos := INC1(pos, max_out); esr_out[pos] := esr_7[cnt]; END_IF;
   END_FOR;
END_IF;
END_FUNCTION_BLOCK

FUNCTION_BLOCK ESR_MON_B8
VAR_INPUT
	s0, s1, s2, s3, s4, s5, s6, s7 : BOOL;
	DT_in : DT;
END_VAR
VAR_INPUT CONSTANT
	a0, a1, a2, a3, a4, a5, a6, a7 : STRING(10);
END_VAR
VAR_OUTPUT
	ESR_Flag : BOOL;
END_VAR
VAR_IN_OUT
	ESR_Out: ARRAY [0..3] OF esr_data;
END_VAR
VAR
	x0, x1, x2, x3, x4, x5, x6, x7 : BOOL;
	tx: TIME;
	cnt : INT;
END_VAR

(* read system timer *)
tx := DWORD_TO_TIME(T_PLC_MS());

ESR_Flag := FALSE;
esr_out[3].typ := 0;
esr_out[2].typ := 0;
esr_out[1].typ := 0;
esr_out[0].typ := 0;
cnt := 0;

(* check if inputs have chaged and fill buffer *)
IF s0 <> X0 THEN
	esr_out[cnt].typ := USINT_TO_BYTE(10 + BOOL_TO_USINT(s0));
	esr_out[cnt].adress := a0;
	esr_out[cnt].DS := DT_in;
	esr_out[cnt].TS := TX;
	X0 := S0;
	cnt := cnt + 1;
	esr_flag := TRUE;
END_IF;
IF s1 <> X1 THEN
	esr_out[cnt].typ := USINT_TO_BYTE(10 + BOOL_TO_USINT(s1));
	esr_out[cnt].adress := a1;
	esr_out[cnt].DS := DT_in;
	esr_out[cnt].TS := TX;
	X1 := S1;
	cnt := cnt + 1;
	esr_flag := TRUE;
END_IF;
IF s2 <> X2 THEN
	esr_out[cnt].typ := USINT_TO_BYTE(10 + BOOL_TO_USINT(s2));
	esr_out[cnt].adress := a2;
	esr_out[cnt].DS := DT_in;
	esr_out[cnt].TS := TX;
	X2 := S2;
	cnt := cnt + 1;
	esr_flag := TRUE;
END_IF;
IF s3 <> X3 THEN
	esr_out[cnt].typ := USINT_TO_BYTE(10 + BOOL_TO_USINT(s3));
	esr_out[cnt].adress := a3;
	esr_out[cnt].DS := DT_in;
	esr_out[cnt].TS := TX;
	X3 := S3;
	cnt := cnt + 1;
	esr_flag := TRUE;
END_IF;
IF s4 <> X4 AND cnt < 4 THEN
	esr_out[cnt].typ := USINT_TO_BYTE(10 + BOOL_TO_USINT(s4));
	esr_out[cnt].adress := a4;
	esr_out[cnt].DS := DT_in;
	esr_out[cnt].TS := TX;
	X4 := S4;
	cnt := cnt + 1;
	esr_flag := TRUE;
END_IF;
IF s5 <> X5  AND cnt < 4 THEN
	esr_out[cnt].typ := USINT_TO_BYTE(10 + BOOL_TO_USINT(s5));
	esr_out[cnt].adress := a5;
	esr_out[cnt].DS := DT_in;
	esr_out[cnt].TS := TX;
	X5 := S5;
	cnt := cnt + 1;
	esr_flag := TRUE;
END_IF;
IF s6 <> X6  AND cnt < 4 THEN
	esr_out[cnt].typ := USINT_TO_BYTE(10 + BOOL_TO_USINT(s6));
	esr_out[cnt].adress := a6;
	esr_out[cnt].DS := DT_in;
	esr_out[cnt].TS := TX;
	X6 := S6;
	cnt := cnt + 1;
	esr_flag := TRUE;
END_IF;
IF s7 <> X7  AND cnt < 4 THEN
	esr_out[cnt].typ := USINT_TO_BYTE(10 + BOOL_TO_USINT(s7));
	esr_out[cnt].adress := a7;
	esr_out[cnt].DS := DT_in;
	esr_out[cnt].TS := TX;
	X7 := S7;
	cnt := cnt + 1;
	esr_flag := TRUE;
END_IF;
END_FUNCTION_BLOCK

// Commented out for beedance: it reads the bits of a REAL as a DWORD, or back, through a pointer; a beedance reference (REF_TO) refers to a variable of its own type.
// FUNCTION_BLOCK ESR_MON_R4
// VAR_INPUT
// 	R0, R1, R2, R3 : REAL;
// 	DT_in : DT;
// END_VAR
// VAR_INPUT CONSTANT
// 	a0, a1, a2, a3 : STRING(10);
// 	s0, s1, s2, s3 : REAL;
// END_VAR
// VAR_OUTPUT
// 	ESR_Flag : BOOL;
// END_VAR
// VAR_IN_OUT
// 	ESR_Out: ARRAY [0..3] OF esr_data;
// END_VAR
// VAR
// 	p0, p1, p2, p3 : REF_TO DWORD;
// 	x0, x1, x2, x3 : REAL;
// 	tx: TIME;
// 	cnt : INT;
// END_VAR
//
// (* read system timer *)
// tx := DWORD_TO_TIME(T_PLC_MS());
// P0 := REF(R0);
// P1 := REF(R1);
// P2 := REF(R2);
// P3 := REF(R3);
//
// ESR_Flag := FALSE;
// esr_out[3].typ := 0;
// esr_out[2].typ := 0;
// esr_out[1].typ := 0;
// esr_out[0].typ := 0;
// cnt := 0;
//
// (* check if inputs have chaged and fill buffer *)
// IF DIFFER(R0,  X0, S0) THEN
// 	esr_out[cnt].typ := 20;
// 	esr_out[cnt].adress := a0;
// 	esr_out[cnt].DS := DT_in;
// 	esr_out[cnt].TS := TX;
// 	esr_out[cnt].data[0] := Byte_of_Dword(P0^,0);
// 	esr_out[cnt].data[1] := Byte_of_Dword(P0^,1);
// 	esr_out[cnt].data[2] := Byte_of_Dword(P0^,2);
// 	esr_out[cnt].data[3] := Byte_of_Dword(P0^,3);
// 	X0 := R0;
// 	cnt := cnt + 1;
// 	esr_flag := TRUE;
// END_IF;
// IF differ(R1,  X1, S1) THEN
// 	esr_out[cnt].typ := 20;
// 	esr_out[cnt].adress := a1;
// 	esr_out[cnt].DS := DT_in;
// 	esr_out[cnt].TS := TX;
// 	esr_out[cnt].data[0] := Byte_of_Dword(P1^,0);
// 	esr_out[cnt].data[1] := Byte_of_Dword(P1^,1);
// 	esr_out[cnt].data[2] := Byte_of_Dword(P1^,2);
// 	esr_out[cnt].data[3] := Byte_of_Dword(P1^,3);
// 	X1 := R1;
// 	cnt := cnt + 1;
// 	esr_flag := TRUE;
// END_IF;
// IF differ(R2,  X2, S2) THEN
// 	esr_out[cnt].typ := 20;
// 	esr_out[cnt].adress := a2;
// 	esr_out[cnt].DS := DT_in;
// 	esr_out[cnt].TS := TX;
// 	esr_out[cnt].data[0] := Byte_of_Dword(P2^,0);
// 	esr_out[cnt].data[1] := Byte_of_Dword(P2^,1);
// 	esr_out[cnt].data[2] := Byte_of_Dword(P2^,2);
// 	esr_out[cnt].data[3] := Byte_of_Dword(P2^,3);
// 	X2 := R2;
// 	cnt := cnt + 1;
// 	esr_flag := TRUE;
// END_IF;
// IF DIFFER(R3,  X3, S3) THEN
// 	esr_out[cnt].typ := 20;
// 	esr_out[cnt].adress := a3;
// 	esr_out[cnt].DS := DT_in;
// 	esr_out[cnt].TS := TX;
// 	esr_out[cnt].data[0] := Byte_of_Dword(P3^,0);
// 	esr_out[cnt].data[1] := Byte_of_Dword(P3^,1);
// 	esr_out[cnt].data[2] := Byte_of_Dword(P3^,2);
// 	esr_out[cnt].data[3] := Byte_of_Dword(P3^,3);
// 	X3 := R3;
// 	cnt := cnt + 1;
// 	esr_flag := TRUE;
// END_IF;
// END_FUNCTION_BLOCK

FUNCTION_BLOCK ESR_MON_X8
VAR_INPUT
	s0, s1, s2, s3, s4, s5, s6, s7 : BYTE;
	DT_in : DT;
	Mode : BYTE := 3;
END_VAR
VAR_INPUT CONSTANT
	a0, a1, a2, a3, a4, a5, a6, a7 : STRING(10);
END_VAR
VAR_OUTPUT
	ESR_Flag : BOOL;
END_VAR
VAR_IN_OUT
	ESR_Out: ARRAY [0..3] OF esr_data;
END_VAR
VAR
	x0, x1, x2, x3, x4, x5, x6, x7 : BYTE;
	tx: TIME;
	cnt : INT;
END_VAR

(* read system timer *)
tx := DWORD_TO_TIME(T_PLC_MS());

ESR_Flag := FALSE;
esr_out[3].typ := 0;
esr_out[2].typ := 0;
esr_out[1].typ := 0;
esr_out[0].typ := 0;
cnt := 0;

(* check if inputs have chaged and fill buffer *)
IF s0 <> X0 AND ((s0 < 100) OR (S0 > 99 AND S0 < 200 AND mode >= 2) OR (S0 > 199 AND mode = 3)) THEN
	esr_out[cnt] := status_to_ESR(s0, a0, DT_in, TX);
	X0 := S0;
	cnt := cnt + 1;
	esr_flag := TRUE;
END_IF;
IF s1 <> X1 AND ((s1 < 100) OR (S1 > 99 AND S1 < 200 AND mode >= 2) OR (S1 > 199 AND mode = 3)) THEN
	esr_out[cnt] := status_to_ESR(s1, a1, DT_in, TX);
	X1 := S1;
	cnt := cnt + 1;
	esr_flag := TRUE;
END_IF;
IF s2 <> X2 AND ((s2 < 100) OR (S2 > 99 AND S2 < 200 AND mode >= 2) OR (S2 > 199 AND mode = 3)) THEN
	esr_out[cnt] := status_to_ESR(s2, a2, DT_in, TX);
	X2 := S2;
	cnt := cnt + 1;
	esr_flag := TRUE;
END_IF;
IF s3 <> X3 AND ((s3 < 100) OR (S3 > 99 AND S3 < 200 AND mode >= 2) OR (S3 > 199 AND mode = 3)) THEN
	esr_out[cnt] := status_to_ESR(s3, a3, DT_in, TX);
	X3 := S3;
	cnt := cnt + 1;
	esr_flag := TRUE;
END_IF;
IF cnt < 4 AND s4 <> X4 AND ((s4 < 100) OR (S4 > 99 AND S4 < 200 AND mode >= 2) OR (S4 > 199 AND mode = 3)) THEN
	esr_out[cnt] := status_to_ESR(s4, a4, DT_in, TX);
	X4 := S4;
	cnt := cnt + 1;
	esr_flag := TRUE;
END_IF;
IF cnt < 4 AND s5 <> X5 AND ((s5 < 100) OR (S5 > 99 AND S5 < 200 AND mode >= 2) OR (S5 > 199 AND mode = 3)) THEN
	esr_out[cnt] := status_to_ESR(s5, a5, DT_in, TX);
	X5 := S5;
	cnt := cnt + 1;
	esr_flag := TRUE;
END_IF;
IF cnt < 4 AND s6 <> X6 AND ((s6 < 100) OR (S6 > 99 AND S6 < 200 AND mode >= 2) OR (S6 > 199 AND mode = 3)) THEN
	esr_out[cnt] := status_to_ESR(s6, a6, DT_in, TX);
	X6 := S6;
	cnt := cnt + 1;
	esr_flag := TRUE;
END_IF;
IF cnt < 4 AND s7 <> X7 AND ((s7 < 100) OR (S7 > 99 AND S7 < 200 AND mode >= 2) OR (S7 > 199 AND mode = 3)) THEN
	esr_out[cnt] := status_to_ESR(s7, a7, DT_in, TX);
	X7 := S7;
	cnt := cnt + 1;
	esr_flag := TRUE;
END_IF;
END_FUNCTION_BLOCK
